        //----------------------------------------------------
        // Paste Position
        //----------------------------------------------------
        GVL_1.DATA_RB_B.X_POS[GVL.HMI_B_PointNoSelected] := GVL.B_PointClipboardX;

        GVL_1.DATA_RB_B.Y_POS[GVL.HMI_B_PointNoSelected] := GVL.B_PointClipboardY;

        GVL_1.DATA_RB_B.Z_POS[GVL.HMI_B_PointNoSelected] := GVL.B_PointClipboardZ;

        GVL_1.DATA_RB_B.R_POS[GVL.HMI_B_PointNoSelected] := GVL.B_PointClipboardR;


//         //----------------------------------------------------
//         // Đồng thời cập nhật vùng Edit để HMI hiển thị
//         // ngay dữ liệu vừa Paste
//         //----------------------------------------------------
//         GVL.HMI_B_Edit_PointNo := GVL.HMI_B_PointNoSelected;
// 
//         GVL.HMI_B_Edit_Pos_Name := GVL.B_PointClipboardName;
// 
//         GVL.HMI_B_Edit_Pos_X := GVL.B_PointClipboardX;
// 
//         GVL.HMI_B_Edit_Pos_Y := GVL.B_PointClipboardY;
// 
//         GVL.HMI_B_Edit_Pos_Z := GVL.B_PointClipboardZ;
// 
//         GVL.HMI_B_Edit_Pos_R := GVL.B_PointClipboardR;

    END_IF;

    //--------------------------------------------------------
    // Không xóa Clipboard.
    //
    // Nhờ vậy có thể:
    // Copy P10 → Paste P20 → Paste P21 → Paste P22...
    //--------------------------------------------------------

    GVL.HMI_B_EditPointReq := 0;

END_IF;

//============================================================
// DELETE ALL POINTS
//
// HMI_A_EditPointReq = 27
//
// Xóa toàn bộ Point Database.
//============================================================

Delete_all_point_B(IN := GVL.HMI_B_EditPointReq_Arr[7], PT := T#2S);
IF Delete_all_point_B.Q THEN

    FOR iPoint := 1 TO 500 DO

        //----------------------------------------------------
        // Clear Name
        //----------------------------------------------------
        GVL_1.Point_Name_B[iPoint] := '';

        //----------------------------------------------------
        // Clear Position
        //----------------------------------------------------
        GVL_1.DATA_RB_B.X_POS[iPoint] := 0.0;
        GVL_1.DATA_RB_B.Y_POS[iPoint] := 0.0;
        GVL_1.DATA_RB_B.Z_POS[iPoint] := 0.0;
        GVL_1.DATA_RB_B.R_POS[iPoint] := 0.0;

    END_FOR;


    //--------------------------------------------------------
    // Clear vùng Edit trên HMI
    //--------------------------------------------------------
    GVL.HMI_B_Edit_PointNo  := 0;
    GVL.HMI_B_Edit_Pos_Name := '';

    GVL.HMI_B_Edit_Pos_X := 0.0;
    GVL.HMI_B_Edit_Pos_Y := 0.0;
    GVL.HMI_B_Edit_Pos_Z := 0.0;
    GVL.HMI_B_Edit_Pos_R := 0.0;


    //--------------------------------------------------------
    // Reset Point đang chọn
    //--------------------------------------------------------
    GVL.HMI_B_PointNoSelected := 0;


    //--------------------------------------------------------
    // Em khuyên KHÔNG xóa Clipboard.
    //
    // Nếu Delete All nhầm, dữ liệu Point vừa Copy vẫn còn
    // và có thể Paste lại.
    //--------------------------------------------------------

    GVL.HMI_B_EditPointReq := 0;
	GVL.HMI_B_EditPointReq_Arr[7] := FALSE;

END_IF;
END_ACTION

END_PROGRAM

// Just_Motion_Control_x86_64_Linux_SM_WV/Application/FC_/RBA/F_EvalCondRowFromEdit_A
FUNCTION F_EvalCondRowFromEdit_A : BOOL
VAR_INPUT
	RowNo : INT;
END_VAR
VAR
	actualValue : DINT;
END_VAR

IF (RowNo < 1) OR (RowNo > 10) THEN
    F_EvalCondRowFromEdit_A := FALSE;
    RETURN;
END_IF;

IF NOT GVL.HMI_A_CondEditRowEnable[RowNo] THEN
    F_EvalCondRowFromEdit_A := TRUE;
    RETURN;
END_IF;

// Đọc giá trị thực tế hiện tại
actualValue := F_GetCondValue_A(
    Source := GVL.HMI_A_CondEditSource[RowNo],
    Index  := GVL.HMI_A_CondEditIndex[RowNo]
);

// Lưu actual value để HMI hiển thị
GVL.HMI_A_CondMonActualValue[RowNo] := actualValue;

// So sánh theo operator
CASE GVL.HMI_A_CondEditOperator[RowNo] OF
    1: F_EvalCondRowFromEdit_A := actualValue = GVL.HMI_A_CondEditSetValue[RowNo];
    2: F_EvalCondRowFromEdit_A := actualValue <> GVL.HMI_A_CondEditSetValue[RowNo];
    3: F_EvalCondRowFromEdit_A := actualValue >  GVL.HMI_A_CondEditSetValue[RowNo];
    4: F_EvalCondRowFromEdit_A := actualValue >= GVL.HMI_A_CondEditSetValue[RowNo];
    5: F_EvalCondRowFromEdit_A := actualValue <  GVL.HMI_A_CondEditSetValue[RowNo];
    6: F_EvalCondRowFromEdit_A := actualValue <= GVL.HMI_A_CondEditSetValue[RowNo];
ELSE
    F_EvalCondRowFromEdit_A := FALSE;
END_CASE;

END_FUNCTION

// Just_Motion_Control_x86_64_Linux_SM_WV/Application/FC_/RBB/F_EvalCondRowFromEdit_B
FUNCTION F_EvalCondRowFromEdit_B : BOOL
VAR_INPUT
	RowNo : INT;
END_VAR
VAR
	actualValue : DINT;
END_VAR

IF (RowNo < 1) OR (RowNo > 10) THEN
    F_EvalCondRowFromEdit_B := FALSE;
    RETURN;
END_IF;

IF NOT GVL.HMI_B_CondEditRowEnable[RowNo] THEN
    F_EvalCondRowFromEdit_B := TRUE;
    RETURN;
END_IF;

// Đọc giá trị thực tế hiện tại
actualValue := F_GetCondValue_B(
    Source := GVL.HMI_B_CondEditSource[RowNo],
    Index  := GVL.HMI_B_CondEditIndex[RowNo]
);

// Lưu actual value để HMI hiển thị
GVL.HMI_B_CondMonActualValue[RowNo] := actualValue;

// So sánh theo operator
CASE GVL.HMI_B_CondEditOperator[RowNo] OF
    1: F_EvalCondRowFromEdit_B := actualValue = GVL.HMI_B_CondEditSetValue[RowNo];
    2: F_EvalCondRowFromEdit_B := actualValue <> GVL.HMI_B_CondEditSetValue[RowNo];
    3: F_EvalCondRowFromEdit_B := actualValue >  GVL.HMI_B_CondEditSetValue[RowNo];
    4: F_EvalCondRowFromEdit_B := actualValue >= GVL.HMI_B_CondEditSetValue[RowNo];
    5: F_EvalCondRowFromEdit_B := actualValue <  GVL.HMI_B_CondEditSetValue[RowNo];
    6: F_EvalCondRowFromEdit_B := actualValue <= GVL.HMI_B_CondEditSetValue[RowNo];
ELSE
    F_EvalCondRowFromEdit_B := FALSE;
END_CASE;

END_FUNCTION

// Just_Motion_Control_x86_64_Linux_SM_WV/Application/PRG_ROBOT/POU_HOMING
PROGRAM POU_HOMING
VAR
	MC_GroupStop_RBA, MC_GroupStop_RBB : MC_GroupStop;
	MC_Stop_A0: MC_Stop;
	MC_Stop_A1: MC_Stop;
	MC_Stop_A2: MC_Stop;
	MC_Stop_A3: MC_Stop;
	MC_GroupSetPosition_RB1: MC_GroupSetPosition;
	Origin_Pos_A: SM3_Robotics.SMC_POS_REF;
	MC_GroupSetPosition_RB2: MC_GroupSetPosition;
	Origin_Pos_B: SM3_Robotics.SMC_POS_REF;
	MC_Stop_B0: MC_Stop;
	MC_Stop_B2: MC_Stop;
	MC_Stop_B1: MC_Stop;
	MC_Stop_B3: MC_Stop;
	MC_Home_A0: MC_Home;
	MC_Home_A1: MC_Home;
	MC_Home_A2: MC_Home;
	MC_Home_A3: MC_Home;
	MC_Home_B0: MC_Home;
	MC_Home_B1: MC_Home;
	MC_Home_B2: MC_Home;
	MC_Home_B3: MC_Home;
	MC_Power_za: MC_Power;
	MC_Jog_za: MC_Jog;
	MC_Power_ZB: MC_Power;
	MC_Jog_ZB: MC_Jog;
	SMC_SetSoftwareLimits_A0: SMC_SetSoftwareLimits;
	SMC_SetSoftwareLimits_A1: SMC_SetSoftwareLimits;
	SMC_SetSoftwareLimits_A2: SMC_SetSoftwareLimits;
	SMC_SetSoftwareLimits_A3: SMC_SetSoftwareLimits;
	SMC_SetSoftwareLimits_B0: SMC_SetSoftwareLimits;
	SMC_SetSoftwareLimits_B1: SMC_SetSoftwareLimits;
	SMC_SetSoftwareLimits_B2: SMC_SetSoftwareLimits;
	SMC_SetSoftwareLimits_B3: SMC_SetSoftwareLimits;
	
	MC_ReadError_A0: MC_ReadAxisError;
	MC_ReadError_A1: MC_ReadAxisError;
	MC_ReadError_A2: MC_ReadAxisError;
	MC_ReadError_A3: MC_ReadAxisError;
	MC_ReadError_B0: MC_ReadAxisError;
	MC_ReadError_B1: MC_ReadAxisError;
	MC_ReadError_B2: MC_ReadAxisError;
	MC_ReadError_B3: MC_ReadAxisError;
	
END_VAR
VAR
	Bit_Stop, BitStop_Tor_A, BitStop_Tor_B, BitStop_TorDiff_A, BitStop_TorDiff_B, BitStop_Error_Axis_RB_A, BitStop_Error_Axis_RB_B : BOOL;	
	//EMG AT %IX1.1 : BOOL;
	
	// Home Z 
	D_HomeZ_RB1, D_HomeZ_RB2 : INT;
	//SS_DOG_Z1 AT %IX1.3 : BOOL;
	//SS_DOG_Z2 AT %IX1.2 : BOOL;
	R_TRIG_Z1, R_TRIG_Z2 : R_TRIG;
	Homing_Z1, Homing_Z2, Home_Done_Z1, Home_Done_Z2 : BOOL;
END_VAR

VAR // SETLMIT
	ENABLE_POWER_A,DISABLE_POWER_A, ENABLE_POWER_B, DISABLE_POWER_B : BYTE;
	
END_VAR
VAR
	TORQUE_ACT_A0 AT %IW40 : INT;
	TORQUE_ACT_A1 AT %IW48 : INT;
	TORQUE_ACT_A2 AT %IW56 : INT;
	TORQUE_ACT_A3 AT %IW64 : INT;
	TORQUE_ACT_B0 AT %IW72 : INT;
	TORQUE_ACT_B1 AT %IW80 : INT;
	TORQUE_ACT_B2 AT %IW88 : INT;
	TORQUE_ACT_B3 AT %IW96 : INT;
	TORQUE_LIMIT_A0, TORQUE_LIMIT_A1, TORQUE_LIMIT_A2, TORQUE_LIMIT_A3 : INT;
	TORQUE_LIMIT_B0, TORQUE_LIMIT_B1, TORQUE_LIMIT_B2, TORQUE_LIMIT_B3 : INT;
	
END_VAR

//namnv0804
VAR
	VEL_ACT_A0 AT %ID19 : DINT;
	VEL_ACT_A1 AT %ID23 : DINT;
	VEL_ACT_A2 AT %ID27 : DINT;
	VEL_ACT_A3 AT %ID31 : DINT;
	VEL_ACT_B0 AT %ID35 : DINT;
	VEL_ACT_B1 AT %ID39 : DINT;
	VEL_ACT_B2 AT %ID43 : DINT;
	VEL_ACT_B3 AT %ID47 : DINT;
	
	VEL_SET_A0 AT %QD118 : DINT;
	VEL_SET_A1 AT %QD122 : DINT;
	VEL_SET_A2 AT %QD126 : DINT;
	VEL_SET_A3 AT %QD130 : DINT;
	VEL_SET_B0 AT %QD134 : DINT;
	VEL_SET_B1 AT %QD138 : DINT;
	VEL_SET_B2 AT %QD142 : DINT;
	VEL_SET_B3 AT %QD146 : DINT;
	
	TorqueDiff_RB_A0, TorqueDiff_RB_A1, TorqueDiff_RB_A2, TorqueDiff_RB_A3 : FB_TorqueDiff;
	TorqueDiff_RB_B0, TorqueDiff_RB_B1, TorqueDiff_RB_B2, TorqueDiff_RB_B3 : FB_TorqueDiff;
	TORQUE_DIFF_LIMIT_B0, TORQUE_DIFF_LIMIT_B1, TORQUE_DIFF_LIMIT_B2, TORQUE_DIFF_LIMIT_B3 : INT;
	TORQUE_DIFF_MAX_A0, TORQUE_DIFF_MAX_A1, TORQUE_DIFF_MAX_A2, TORQUE_DIFF_MAX_A3 : INT;
	TORQUE_DIFF_MAX_B0, TORQUE_DIFF_MAX_B1, TORQUE_DIFF_MAX_B2, TORQUE_DIFF_MAX_B3 : INT;
	TORQUE_DIFF_MIN_A0, TORQUE_DIFF_MIN_A1, TORQUE_DIFF_MIN_A2, TORQUE_DIFF_MIN_A3 : INT;
	TORQUE_DIFF_MIN_B0, TORQUE_DIFF_MIN_B1, TORQUE_DIFF_MIN_B2, TORQUE_DIFF_MIN_B3 : INT;
	
	VEL_MAX_A0, VEL_MAX_A1, VEL_MAX_A2, VEL_MAX_A3 : DINT;
	VEL_MAX_B0, VEL_MAX_B1, VEL_MAX_B2, VEL_MAX_B3 : DINT;
	
	VEL_SET_MAX_A0, VEL_SET_MAX_A1, VEL_SET_MAX_A2, VEL_SET_MAX_A3 : DINT;
	VEL_SET_MAX_B0, VEL_SET_MAX_B1, VEL_SET_MAX_B2, VEL_SET_MAX_B3 : DINT;
	Vel_Act_Per_Vel_Set_A0, Vel_Act_Per_Vel_Set_A1, Vel_Act_Per_Vel_Set_A2, Vel_Act_Per_Vel_Set_A3: INT;
	Vel_Act_Per_Vel_Set_B0, Vel_Act_Per_Vel_Set_B1, Vel_Act_Per_Vel_Set_B2, Vel_Act_Per_Vel_Set_B3: INT;
	Torque_arr_A0 : ARRAY[0..20000] OF INT;
	i_A0 : INT := 0;
END_VAR
VAR // added by the converter: edge detectors and wires of the graphical bodies
    _w1, _w2, _w3, _w4, _w5, _w6, _w7, _w8 : LREAL;
END_VAR

// namnv3103
// TORQUE_LIMIT_A0:= 3600;
// TORQUE_LIMIT_A1:= 2500;
// TORQUE_LIMIT_A2:= 2000;
// TORQUE_LIMIT_A3:= 2000;
// 
// TORQUE_LIMIT_B0:= 3600;
// TORQUE_LIMIT_B1:= 2500;
// TORQUE_LIMIT_B2:= 2000;
// TORQUE_LIMIT_B3:= 2000;

TORQUE_LIMIT_A0:= GVL.Pro4_.Auto.TORQUE_LIMIT_SET_A0;
TORQUE_LIMIT_A1:= GVL.Pro4_.Auto.TORQUE_LIMIT_SET_A1;
TORQUE_LIMIT_A2:= GVL.Pro4_.Auto.TORQUE_LIMIT_SET_A2;
TORQUE_LIMIT_A3:= GVL.Pro4_.Auto.TORQUE_LIMIT_SET_A3;

TORQUE_LIMIT_B0:= GVL.Pro4_.Auto.TORQUE_LIMIT_SET_B0;
TORQUE_LIMIT_B1:= GVL.Pro4_.Auto.TORQUE_LIMIT_SET_B1;
TORQUE_LIMIT_B2:= GVL.Pro4_.Auto.TORQUE_LIMIT_SET_B2;
TORQUE_LIMIT_B3:= GVL.Pro4_.Auto.TORQUE_LIMIT_SET_B3;

IF GVL.Reset_Torque_Max THEN
	GVL.Torque_Max.A0 := 0;
	GVL.Torque_Max.A1 := 0;
	GVL.Torque_Max.A2 := 0;
	GVL.Torque_Max.A3 := 0;
	GVL.Torque_Max.B0 := 0;
	GVL.Torque_Max.B1 := 0;
	GVL.Torque_Max.B2 := 0;
	GVL.Torque_Max.B3 := 0;
	TORQUE_DIFF_MAX_A0 := 0;
	TORQUE_DIFF_MAX_A1 := 0;
	TORQUE_DIFF_MAX_A2 := 0;
	TORQUE_DIFF_MAX_A3 := 0;
	TORQUE_DIFF_MAX_B0 := 0;
	TORQUE_DIFF_MAX_B1 := 0;
	TORQUE_DIFF_MAX_B2 := 0;
	TORQUE_DIFF_MAX_B3 := 0;
	VEL_MAX_A0 := 0;
	VEL_MAX_A1 := 0;
	VEL_MAX_A2 := 0;
	VEL_MAX_A3 := 0;
	VEL_MAX_B0 := 0;
	VEL_MAX_B1 := 0;
	VEL_MAX_B2 := 0;
	VEL_MAX_B3 := 0;
	VEL_SET_MAX_A0 := 0;
END_IF
GVL.Torque_Max.A0 := MAX(ABS(TORQUE_ACT_A0), GVL.Torque_Max.A0);
GVL.Torque_Max.A1 := MAX(ABS(TORQUE_ACT_A1), GVL.Torque_Max.A1);
GVL.Torque_Max.A2 := MAX(ABS(TORQUE_ACT_A2), GVL.Torque_Max.A2);
GVL.Torque_Max.A3 := MAX(ABS(TORQUE_ACT_A3), GVL.Torque_Max.A3);

GVL.Torque_Max.B0 := MAX(ABS(TORQUE_ACT_B0), GVL.Torque_Max.B0);
GVL.Torque_Max.B1 := MAX(ABS(TORQUE_ACT_B1), GVL.Torque_Max.B1);
GVL.Torque_Max.B2 := MAX(ABS(TORQUE_ACT_B2), GVL.Torque_Max.B2);
GVL.Torque_Max.B3 := MAX(ABS(TORQUE_ACT_B3), GVL.Torque_Max.B3);

// IF (ABS(TORQUE_ACT_A0) > TORQUE_LIMIT_A0) OR (ABS(TORQUE_ACT_A1) > TORQUE_LIMIT_A1) OR (ABS(TORQUE_ACT_A2) > TORQUE_LIMIT_A2) OR (ABS(TORQUE_ACT_A3) > TORQUE_LIMIT_A3) THEN
// 	BitStop_Tor_A := TRUE;
// ELSE
// 	BitStop_Tor_A := FALSE;
// END_IF
// 
// IF (ABS(TORQUE_ACT_B0) > TORQUE_LIMIT_B0) OR (ABS(TORQUE_ACT_B1) > TORQUE_LIMIT_B1) OR (ABS(TORQUE_ACT_B2) > TORQUE_LIMIT_B2) OR (ABS(TORQUE_ACT_B3) > TORQUE_LIMIT_B3) THEN
// 	BitStop_Tor_B := TRUE;
// ELSE
// 	BitStop_Tor_B := FALSE;
// END_IF

//namnv0804

VEL_MAX_A0 := MAX(VEL_MAX_A0, ABS(VEL_ACT_A0));
VEL_MAX_A1 := MAX(VEL_MAX_A1, ABS(VEL_ACT_A1));
VEL_MAX_A2 := MAX(VEL_MAX_A2, ABS(VEL_ACT_A2));
VEL_MAX_A3 := MAX(VEL_MAX_A3, ABS(VEL_ACT_A3));
VEL_MAX_B0 := MAX(VEL_MAX_B0, ABS(VEL_ACT_B0));
VEL_MAX_B1 := MAX(VEL_MAX_B1, ABS(VEL_ACT_B1));
VEL_MAX_B2 := MAX(VEL_MAX_B2, ABS(VEL_ACT_B2));
VEL_MAX_B3 := MAX(VEL_MAX_B3, ABS(VEL_ACT_B3));
VEL_SET_MAX_A0 := MAX(VEL_SET_MAX_A0, ABS(VEL_SET_A0));
Vel_Act_Per_Vel_Set_A0 := LREAL_TO_INT(
    (DINT_TO_LREAL(VEL_ACT_A0) * 100.0) / DINT_TO_LREAL(VEL_SET_A0)
);
Vel_Act_Per_Vel_Set_A1 := LREAL_TO_INT(
    (DINT_TO_LREAL(VEL_ACT_A1) * 100.0) / DINT_TO_LREAL(VEL_SET_A1)
);
Vel_Act_Per_Vel_Set_A2 := LREAL_TO_INT(
    (DINT_TO_LREAL(VEL_ACT_A2) * 100.0) / DINT_TO_LREAL(VEL_SET_A2)
);
Vel_Act_Per_Vel_Set_A3 := LREAL_TO_INT(
    (DINT_TO_LREAL(VEL_ACT_A3) * 100.0) / DINT_TO_LREAL(VEL_SET_A3)
);
Vel_Act_Per_Vel_Set_B0 := LREAL_TO_INT(
    (DINT_TO_LREAL(VEL_ACT_B0) * 100.0) / DINT_TO_LREAL(VEL_SET_B0)
);
Vel_Act_Per_Vel_Set_B1 := LREAL_TO_INT(
    (DINT_TO_LREAL(VEL_ACT_B1) * 100.0) / DINT_TO_LREAL(VEL_SET_B1)
);
Vel_Act_Per_Vel_Set_B2 := LREAL_TO_INT(
    (DINT_TO_LREAL(VEL_ACT_B2) * 100.0) / DINT_TO_LREAL(VEL_SET_B2)
);
Vel_Act_Per_Vel_Set_B3 := LREAL_TO_INT(
    (DINT_TO_LREAL(VEL_ACT_B3) * 100.0) / DINT_TO_LREAL(VEL_SET_B3)
);

TorqueDiff_RB_A0(
	Enable := TRUE,
	TorqueNow := TORQUE_ACT_A0,
	PercentVel := Vel_Act_Per_Vel_Set_A0,
	Threshold := 400,
	CycleTime_s := 0.01
);
TorqueDiff_RB_A1(
	Enable := TRUE,
	TorqueNow := TORQUE_ACT_A1,
	PercentVel := Vel_Act_Per_Vel_Set_A1,
	Threshold := 500,
	CycleTime_s := 0.01
);
TorqueDiff_RB_A2(
	Enable := TRUE,
	TorqueNow := TORQUE_ACT_A2,
	PercentVel := Vel_Act_Per_Vel_Set_A2,
	Threshold := 500,
	CycleTime_s := 0.01
);
TorqueDiff_RB_A3(
	Enable := TRUE,
	TorqueNow := TORQUE_ACT_A3,
	PercentVel := Vel_Act_Per_Vel_Set_A3,
	Threshold := 100,
	CycleTime_s := 0.01
);

TorqueDiff_RB_B0(
	Enable := TRUE,
	TorqueNow := TORQUE_ACT_B0,
	PercentVel := Vel_Act_Per_Vel_Set_B0,
	Threshold := 500,
	CycleTime_s := 0.01
);
TorqueDiff_RB_B1(
	Enable := TRUE,
	TorqueNow := TORQUE_ACT_B1,
	PercentVel := Vel_Act_Per_Vel_Set_B1,
	Threshold := 500,
	CycleTime_s := 0.01
);
TorqueDiff_RB_B2(
	Enable := TRUE,
	TorqueNow := TORQUE_ACT_B2,
	PercentVel := Vel_Act_Per_Vel_Set_B2,
	Threshold := 500,
	CycleTime_s := 0.01
);
TorqueDiff_RB_B3(
	Enable := TRUE,
	TorqueNow := TORQUE_ACT_B3,
	PercentVel := Vel_Act_Per_Vel_Set_B3,
	Threshold := 100,
	CycleTime_s := 0.01
);

TORQUE_DIFF_MAX_A0 := MAX(TORQUE_DIFF_MAX_A0, TorqueDiff_RB_A0.AbsDeltaTorque);
TORQUE_DIFF_MAX_A1 := MAX(TORQUE_DIFF_MAX_A1, TorqueDiff_RB_A1.AbsDeltaTorque);
TORQUE_DIFF_MAX_A2 := MAX(TORQUE_DIFF_MAX_A2, TorqueDiff_RB_A2.AbsDeltaTorque);
TORQUE_DIFF_MAX_A3 := MAX(TORQUE_DIFF_MAX_A3, TorqueDiff_RB_A3.AbsDeltaTorque);
TORQUE_DIFF_MAX_B0 := MAX(TORQUE_DIFF_MAX_B0, TorqueDiff_RB_B0.AbsDeltaTorque);
TORQUE_DIFF_MAX_B1 := MAX(TORQUE_DIFF_MAX_B1, TorqueDiff_RB_B1.AbsDeltaTorque);
TORQUE_DIFF_MAX_B2 := MAX(TORQUE_DIFF_MAX_B2, TorqueDiff_RB_B2.AbsDeltaTorque);
TORQUE_DIFF_MAX_B3 := MAX(TORQUE_DIFF_MAX_B3, TorqueDiff_RB_B3.AbsDeltaTorque);

IF (TorqueDiff_RB_A0.Alarm) OR (TorqueDiff_RB_A1.Alarm) OR (TorqueDiff_RB_A2.Alarm) OR (TorqueDiff_RB_A3.Alarm) THEN
	BitStop_TorDiff_A := TRUE;
ELSE
	BitStop_TorDiff_A := FALSE;
END_IF

IF (TorqueDiff_RB_B0.Alarm) OR (TorqueDiff_RB_B1.Alarm) OR (TorqueDiff_RB_B2.Alarm) OR (TorqueDiff_RB_B3.Alarm) THEN
	BitStop_TorDiff_B := TRUE;
ELSE
	BitStop_TorDiff_B := FALSE;
END_IF


ACT_HOMING();
ACT_STOP();
ACT_Home_Z();
ACT_SETLIMIT();
ACT_ERROR(); //namnv0304

//Origin_Pos_A.c.X := 550;
//Origin_Pos_B.c.X := 0;
//Origin_Pos_B.a.a0 := 0;

ACTION ACT_ERROR:
MC_ReadError_A0(Axis := A0, Enable := A0.bError); // MC_ReadAxisError
MC_ReadError_B0(Axis := B0, Enable := B0.bError); // MC_ReadAxisError
MC_ReadError_A2(Axis := A2, Enable := A2.bError); // MC_ReadAxisError
MC_ReadError_B1(Axis := B1, Enable := B1.bError); // MC_ReadAxisError
MC_ReadError_A3(Axis := A3, Enable := A3.bError); // MC_ReadAxisError
MC_ReadError_A1(Axis := A1, Enable := A1.bError); // MC_ReadAxisError
MC_ReadError_B2(Axis := B2, Enable := B2.bError); // MC_ReadAxisError
MC_ReadError_B3(Axis := B3, Enable := B3.bError); // MC_ReadAxisError
END_ACTION

ACTION ACT_Home_Z:
IF GVL.RB_A.M3 AND GVL.RB_A.Manual AND MC_Power_za.Status THEN
	Homing_Z1 := TRUE;
ELSIF NOT GVL.X[9] OR NOT MC_Power_za.Status THEN
	Homing_Z1 := FALSE;
END_IF
MC_Home_A2.Execute := GVL.RB_A.ORG_M3;
/// PRocess
IF Homing_Z1 THEN
CASE D_HomeZ_RB1 OF
	0:
		IF  GVL.X[3] THEN
			MC_Jog_za.Velocity := 10;
			MC_Jog_za.JogBackward := TRUE;
		ELSE
			MC_Jog_za.JogBackward := FALSE;
			D_HomeZ_RB1 := D_HomeZ_RB1 + 10;
		END_IF
	10:
		IF NOT GVL.X[3] THEN
			MC_Jog_za.Velocity := 5;
			MC_Jog_za.JogForward := TRUE;
		ELSE
			D_HomeZ_RB1 := D_HomeZ_RB1 + 5;
		END_IF
	15:
		IF GVL.X[3] THEN
			MC_Jog_za.JogForward := FALSE;
			D_HomeZ_RB1 := D_HomeZ_RB1 + 5;
		END_IF
	20:
		MC_Jog_za.JogForward := FALSE;
		MC_Jog_za.JogBackward := FALSE;
		MC_Home_A2.Execute := TRUE;
		D_HomeZ_RB1 := D_HomeZ_RB1 + 10;
	30:
		IF MC_Home_A2.Done OR MC_Home_A2.Busy THEN
			MC_Home_A2.Execute := FALSE;
			D_HomeZ_RB1 := D_HomeZ_RB1 + 10;
		ELSIF MC_Home_A2.Error THEN
			D_HomeZ_RB1 := 900;
		END_IF					
	40:	
		D_HomeZ_RB1 := D_HomeZ_RB1 + 10;	
	50:
		D_HomeZ_RB1 := 900;
///////////////////////////////////////// Process Done ////////////////////////////////////
	900:
		Homing_Z1 := FALSE;
END_CASE
ELSE
	MC_Jog_za.JogForward := FALSE;
	MC_Jog_za.JogBackward := FALSE;
	D_HomeZ_RB1 := 0;
END_IF



///// Home Z2 robot B

IF GVL.RB_B.M3 AND GVL.RB_B.Manual AND MC_Power_zB.Status THEN
	Homing_Z2 := TRUE;
ELSIF NOT GVL.X[9] OR NOT MC_Power_ZB.Status THEN
	Homing_Z2 := FALSE;
END_IF
MC_Home_B2.Execute := GVL.RB_B.ORG_M3;
/// PRocess
IF Homing_Z2 THEN
CASE D_HomeZ_RB2 OF
	0:
		IF  GVL.X[2] THEN
			MC_Jog_ZB.Velocity := 10;
			MC_Jog_ZB.JogBackward := TRUE;
		ELSE
			MC_Jog_ZB.JogBackward := FALSE;
			D_HomeZ_RB2 := D_HomeZ_RB2 + 10;
		END_IF
	10:
		IF NOT GVL.X[2] THEN
			MC_Jog_ZB.Velocity := 5;
			MC_Jog_ZB.JogForward := TRUE;
		ELSE
			D_HomeZ_RB2 := D_HomeZ_RB2 + 5;
		END_IF
	15:
		IF GVL.X[2] THEN
			MC_Jog_ZB.JogForward := FALSE;
			D_HomeZ_RB2 := D_HomeZ_RB2 + 5;
		END_IF
	20:
		MC_Jog_ZB.JogForward := FALSE;
		MC_Jog_ZB.JogBackward := FALSE;
		MC_Home_b2.Execute := TRUE;
		D_HomeZ_RB2 := D_HomeZ_RB2 + 10;
	30:
		IF MC_Home_b2.Done OR MC_Home_b2.Busy THEN
			MC_Home_b2.Execute := FALSE;
			D_HomeZ_RB2 := D_HomeZ_RB2 + 10;
		ELSIF MC_Home_b2.Error THEN
			D_HomeZ_RB2 := 900;
		END_IF					
	40:	
		D_HomeZ_RB2 := D_HomeZ_RB2 + 10;	
	50:
		D_HomeZ_RB2 := 900;
///////////////////////////////////////// Process Done ////////////////////////////////////
	900:
		Homing_Z2 := FALSE;
END_CASE
ELSE
	MC_Jog_ZB.JogForward := FALSE;
	MC_Jog_ZB.JogBackward := FALSE;
	D_HomeZ_RB2 := 0;
END_IF
END_ACTION

ACTION ACT_HOMING:
MC_GroupSetPosition_RB1(AxisGroup := SCARA_A, Position := Origin_Pos_A, CoordSystem := GVL.RB_A.COORD); // MC_GroupSetPosition
MC_GroupSetPosition_RB2(AxisGroup := SCARA_B, Position := Origin_Pos_B, CoordSystem := GVL.RB_B.COORD); // MC_GroupSetPosition
MC_Power_ZB(Axis := B2); // MC_Power
MC_Jog_za(Axis := A2, Acceleration := 500, Deceleration := 500, Jerk := 1000); // MC_Jog
MC_Jog_ZB(Axis := B2, Acceleration := 500, Deceleration := 500, Jerk := 1000); // MC_Jog
MC_Home_B2(Axis := B2, Position := 0); // MC_Home
MC_Home_A2(Axis := A2, Position := 0); // MC_Home
MC_Home_B1(Axis := B1, Execute := GVL.RB_B.ORG_M2, Position := 0); // MC_Home
MC_Power_za(Axis := A2); // MC_Power
MC_Home_A1(Axis := A1, Execute := GVL.RB_A.ORG_M2, Position := 0); // MC_Home
MC_Home_B3(Axis := B3, Execute := GVL.RB_B.ORG_M4, Position := 0); // MC_Home
MC_Home_A3(Axis := A3, Execute := GVL.RB_A.ORG_M4, Position := 0); // MC_Home
MC_Home_B0(Axis := B0, Execute := GVL.RB_B.ORG_M1, Position := 0); // MC_Home
MC_Home_A0(Axis := A0, Execute := GVL.RB_A.ORG_M1, Position := 0); // MC_Home
MC_Stop_B0(Axis := B0, Deceleration := 100, Jerk := 0); // MC_Stop
MC_Stop_B1(Axis := B1, Deceleration := 100, Jerk := 0); // MC_Stop
MC_Stop_B2(Axis := B2, Deceleration := 100, Jerk := 0); // MC_Stop
MC_Stop_B3(Axis := B3, Deceleration := 100, Jerk := 0); // MC_Stop
MC_Stop_A0(Axis := A0, Deceleration := 100, Jerk := 0); // MC_Stop
MC_Stop_A3(Axis := A3, Deceleration := 100, Jerk := 0); // MC_Stop
MC_Stop_A2(Axis := A2, Deceleration := 100, Jerk := 0); // MC_Stop
MC_Stop_A1(Axis := A1, Deceleration := 100, Jerk := 0); // MC_Stop
END_ACTION

ACTION ACT_SETLIMIT:
_w1 := TO_LREAL(GVL_1.DATA_RB_A.LIMIT_M1_BW);
_w2 := TO_LREAL(GVL_1.DATA_RB_B.LIMIT_M2_FW);
_w3 := TO_LREAL(GVL_1.DATA_RB_B.LIMIT_M2_BW);
SMC_SetSoftwareLimits_A1(
    Axis := A1,
    SWL_Positive := TO_LREAL(GVL_1.DATA_RB_A.LIMIT_M2_FW),
    SWL_Negative := TO_LREAL(GVL_1.DATA_RB_A.LIMIT_M2_BW),
    SWL_Error_Deceleration := 1000,
    SWL_Error_MaxDistance := 10); // SMC_SetSoftwareLimits
_w4 := TO_LREAL(GVL_1.DATA_RB_B.LIMIT_M3_FW);
_w5 := TO_LREAL(GVL_1.DATA_RB_B.LIMIT_M3_BW);
SMC_SetSoftwareLimits_A2(
    Axis := A2,
    SWL_Positive := TO_LREAL(GVL_1.DATA_RB_A.LIMIT_M3_FW),
    SWL_Negative := TO_LREAL(GVL_1.DATA_RB_A.LIMIT_M3_BW),
    SWL_Error_Deceleration := 1000,
    SWL_Error_MaxDistance := 10); // SMC_SetSoftwareLimits
_w6 := TO_LREAL(GVL_1.DATA_RB_B.LIMIT_M4_FW);
_w7 := TO_LREAL(GVL_1.DATA_RB_B.LIMIT_M4_BW);
_w8 := TO_LREAL(GVL_1.DATA_RB_B.LIMIT_M1_FW);
SMC_SetSoftwareLimits_A3(
    Axis := A3,
    SWL_Positive := TO_LREAL(GVL_1.DATA_RB_A.LIMIT_M4_FW),
    SWL_Negative := TO_LREAL(GVL_1.DATA_RB_A.LIMIT_M4_BW),
    SWL_Error_Deceleration := 1000,
    SWL_Error_MaxDistance := 10); // SMC_SetSoftwareLimits
SMC_SetSoftwareLimits_B0(
    Axis := B0,
    SWL_Positive := _w8,
    SWL_Negative := TO_LREAL(GVL_1.DATA_RB_B.LIMIT_M1_BW),
    SWL_Error_Deceleration := 1000,
    SWL_Error_MaxDistance := 10); // SMC_SetSoftwareLimits
SMC_SetSoftwareLimits_B2(
    Axis := B2,
    SWL_Positive := _w4,
    SWL_Negative := _w5,
    SWL_Error_Deceleration := 1000,
    SWL_Error_MaxDistance := 10); // SMC_SetSoftwareLimits
SMC_SetSoftwareLimits_B3(
    Axis := B3,
    SWL_Positive := _w6,
    SWL_Negative := _w7,
    SWL_Error_Deceleration := 1000,
    SWL_Error_MaxDistance := 10); // SMC_SetSoftwareLimits
SMC_SetSoftwareLimits_A0(
    Axis := A0,
    SWL_Positive := TO_LREAL(GVL_1.DATA_RB_A.LIMIT_M1_FW),
    SWL_Negative := _w1,
    SWL_Error_Deceleration := 1000,
    SWL_Error_MaxDistance := 10); // SMC_SetSoftwareLimits
SMC_SetSoftwareLimits_B1(
    Axis := B1,
    SWL_Positive := _w2,
    SWL_Negative := _w3,
    SWL_Error_Deceleration := 1000,
    SWL_Error_MaxDistance := 10); // SMC_SetSoftwareLimits
END_ACTION

ACTION ACT_STOP:
IF (MC_ReadError_A0.AxisError OR MC_ReadError_A1.AxisError OR MC_ReadError_A2.AxisError OR MC_ReadError_A3.AxisError) 
OR (MC_ReadError_A0.Error OR MC_ReadError_A1.Error OR MC_ReadError_A2.Error OR MC_ReadError_A3.Error)
OR A0.bError OR A1.bError OR A2.bError OR A3.bError THEN
	BitStop_Error_Axis_RB_A := TRUE;
ELSE
	BitStop_Error_Axis_RB_A := FALSE;
END_IF

IF (MC_ReadError_B0.AxisError OR MC_ReadError_B1.AxisError OR MC_ReadError_B2.AxisError OR MC_ReadError_B3.AxisError) 
OR (MC_ReadError_B0.Error OR MC_ReadError_B1.Error OR MC_ReadError_B2.Error OR MC_ReadError_B3.Error) 
OR B0.bError OR B1.bError OR B2.bError OR B3.bError THEN
	BitStop_Error_Axis_RB_B := TRUE;
ELSE
	BitStop_Error_Axis_RB_B := FALSE;
END_IF

IF Bit_Stop = TRUE OR NOT GVL.X[9] OR BitStop_Tor_A OR BitStop_Error_Axis_RB_A 
OR GVL.RB_Signal_In.HMI_STOP OR NOT GVL.RB_Signal_In.HMI_EMG OR GVL.A_RunStop 
OR POU_MONITOR_ROBOT.MC_GroupReadStatus_RBA.Error OR GVL.RB_A_.ERROR
OR SCARA_A.m_group_error > 0 THEN
	MC_Stop_A0.Execute:= TRUE;
	MC_Stop_A1.Execute:= TRUE;
	MC_Stop_A2.Execute:= TRUE;
	MC_Stop_A3.Execute:= TRUE;
	MC_GroupStop_RBA.Execute := TRUE;
ELSE
	MC_Stop_A0.Execute:= FALSE;
	MC_Stop_A1.Execute:= FALSE;
	MC_Stop_A2.Execute:= FALSE;
	MC_Stop_A3.Execute:= FALSE;
	MC_GroupStop_RBA.Execute := FALSE;
END_IF

IF Bit_Stop = TRUE OR NOT GVL.X[9] OR BitStop_Tor_B OR BitStop_Error_Axis_RB_B 
OR GVL.RB_Signal_In.HMI_STOP OR NOT GVL.RB_Signal_In.HMI_EMG 
OR POU_MONITOR_ROBOT.MC_GroupReadStatus_RBB.Error OR GVL.RB_B_.ERROR
OR SCARA_B.m_group_error > 0  THEN
	MC_Stop_B0.Execute:= TRUE;
	MC_Stop_B1.Execute:= TRUE;
	MC_Stop_B2.Execute:= TRUE;
	MC_Stop_B3.Execute:= TRUE;
	MC_GroupStop_RBB.Execute := TRUE;
ELSE
	MC_Stop_B0.Execute:= FALSE;
	MC_Stop_B1.Execute:= FALSE;
	MC_Stop_B2.Execute:= FALSE;
	MC_Stop_B3.Execute:= FALSE;
	MC_GroupStop_RBA.Execute := FALSE;
END_IF




/// Condition SoftLimit

IF GVL_1.DATA_RB_A.ENABLE_SOFT_LIMIT THEN
	DISABLE_POWER_A := 0;
	CASE ENABLE_POWER_A OF
		0:
			SMC_SetSoftwareLimits_A0.SWL_Activated := TRUE;
			SMC_SetSoftwareLimits_A1.SWL_Activated := TRUE;
			SMC_SetSoftwareLimits_A2.SWL_Activated := TRUE;
			SMC_SetSoftwareLimits_A3.SWL_Activated := TRUE;
			ENABLE_POWER_A := ENABLE_POWER_A + 5;
		5:
			SMC_SetSoftwareLimits_A0.bExecute := TRUE;
			SMC_SetSoftwareLimits_A1.bExecute := TRUE;
			SMC_SetSoftwareLimits_A2.bExecute := TRUE;
			SMC_SetSoftwareLimits_A3.bExecute := TRUE;
			ENABLE_POWER_A := ENABLE_POWER_A + 5;
		10:
			// DONE	
	END_CASE
ELSE
	ENABLE_POWER_A := 0;
	CASE DISABLE_POWER_A OF
		0:
			SMC_SetSoftwareLimits_A0.bExecute := FALSE;
			SMC_SetSoftwareLimits_A1.bExecute := FALSE;
			SMC_SetSoftwareLimits_A2.bExecute := FALSE;
			SMC_SetSoftwareLimits_A3.bExecute := FALSE;
			DISABLE_POWER_A := DISABLE_POWER_A + 5;
		5:
			SMC_SetSoftwareLimits_A0.SWL_Activated := FALSE;
			SMC_SetSoftwareLimits_A1.SWL_Activated := FALSE;
			SMC_SetSoftwareLimits_A2.SWL_Activated := FALSE;
			SMC_SetSoftwareLimits_A3.SWL_Activated := FALSE;
			DISABLE_POWER_A := DISABLE_POWER_A + 5;
		10:
			SMC_SetSoftwareLimits_A0.bExecute := TRUE;
			SMC_SetSoftwareLimits_A1.bExecute := TRUE;
			SMC_SetSoftwareLimits_A2.bExecute := TRUE;
			SMC_SetSoftwareLimits_A3.bExecute := TRUE;
			DISABLE_POWER_A := DISABLE_POWER_A + 5;			
		15:
			SMC_SetSoftwareLimits_A0.bExecute := FALSE;
			SMC_SetSoftwareLimits_A1.bExecute := FALSE;
			SMC_SetSoftwareLimits_A2.bExecute := FALSE;
			SMC_SetSoftwareLimits_A3.bExecute := FALSE;				
	END_CASE
END_IF;

/// rbB
IF GVL_1.DATA_RB_B.ENABLE_SOFT_LIMIT THEN
	DISABLE_POWER_B:= 0;
	CASE ENABLE_POWER_B OF
		0:
			SMC_SetSoftwareLimits_B0.SWL_Activated := TRUE;
			SMC_SetSoftwareLimits_B1.SWL_Activated := TRUE;
			SMC_SetSoftwareLimits_B2.SWL_Activated := TRUE;
			SMC_SetSoftwareLimits_B3.SWL_Activated := TRUE;
			ENABLE_POWER_B := ENABLE_POWER_B + 5;
		5:
			SMC_SetSoftwareLimits_B0.bExecute := TRUE;
			SMC_SetSoftwareLimits_B1.bExecute := TRUE;
			SMC_SetSoftwareLimits_B2.bExecute := TRUE;
			SMC_SetSoftwareLimits_B3.bExecute := TRUE;
			ENABLE_POWER_B := ENABLE_POWER_B + 5;
		10:
			// DONE	
	END_CASE
ELSE
	ENABLE_POWER_B := 0;
	CASE DISABLE_POWER_B OF
		0:
			SMC_SetSoftwareLimits_B0.bExecute := FALSE;
			SMC_SetSoftwareLimits_B1.bExecute := FALSE;
			SMC_SetSoftwareLimits_B2.bExecute := FALSE;
			SMC_SetSoftwareLimits_B3.bExecute := FALSE;
			DISABLE_POWER_B := DISABLE_POWER_B + 5;
		5:
			SMC_SetSoftwareLimits_B0.SWL_Activated := FALSE;
			SMC_SetSoftwareLimits_B1.SWL_Activated := FALSE;
			SMC_SetSoftwareLimits_B2.SWL_Activated := FALSE;
			SMC_SetSoftwareLimits_B3.SWL_Activated := FALSE;
			DISABLE_POWER_B := DISABLE_POWER_B + 5;
		10:
			SMC_SetSoftwareLimits_B0.bExecute := TRUE;
			SMC_SetSoftwareLimits_B1.bExecute := TRUE;
			SMC_SetSoftwareLimits_B2.bExecute := TRUE;
			SMC_SetSoftwareLimits_B3.bExecute := TRUE;
			DISABLE_POWER_B := DISABLE_POWER_B + 5;			
		15:
			SMC_SetSoftwareLimits_B0.bExecute := FALSE;
			SMC_SetSoftwareLimits_B1.bExecute := FALSE;
			SMC_SetSoftwareLimits_B2.bExecute := FALSE;
			SMC_SetSoftwareLimits_B3.bExecute := FALSE;				
	END_CASE
END_IF;
END_ACTION

END_PROGRAM

// Just_Motion_Control_x86_64_Linux_SM_WV/Application/FB_/FB_TorqueDiff
FUNCTION_BLOCK PUBLIC FB_TorqueDiff
VAR_INPUT
	Enable          : BOOL;
    TorqueNow       : INT;
	PercentVel		: INT;
    Threshold       : INT;
    CycleTime_s     : LREAL;
END_VAR
VAR_OUTPUT
	DeltaTorque     : INT;
    AbsDeltaTorque  : INT;
    TorqueSlope     : LREAL;
    Alarm           : BOOL;
END_VAR
VAR
	TorqueOld       : INT;
	VelOld			: DINT;
    FirstScan       : BOOL := TRUE;
END_VAR

// IF NOT Enable THEN
//     Alarm := FALSE;
//     DeltaTorque := 0;
//     AbsDeltaTorque := 0;
//     TorqueSlope := 0.0;
//     FirstScan := TRUE;
//     RETURN;
// END_IF;

IF FirstScan THEN
    TorqueOld := TorqueNow;
    DeltaTorque := 0;
    AbsDeltaTorque := 0;
    TorqueSlope := 0.0;
    Alarm := FALSE;
    FirstScan := FALSE;
    RETURN;
END_IF;
IF (PercentVel > 70) THEN
	DeltaTorque := TorqueNow - TorqueOld;
	AbsDeltaTorque := ABS(DeltaTorque);
END_IF;

// IF CycleTime_s > 0.0 THEN
//     TorqueSlope := DeltaTorque / CycleTime_s;
// ELSE
//     TorqueSlope := 0.0;
// END_IF;

Alarm := (AbsDeltaTorque > Threshold);

TorqueOld := TorqueNow;

END_FUNCTION_BLOCK

// Just_Motion_Control_x86_64_Linux_SM_WV/Application/PRG_ROBOT/PRG_TrackingObjectSource_A
PROGRAM PRG_TrackingObjectSource_A
VAR
    fbSensorSourceA : ARRAY[1..GVL.C_MAX_SENSOR_SOURCES] OF FB_SensorObjectSource;
    uiSensorSource : UINT;
	fbVisionSourceA : ARRAY[1..GVL.C_MAX_VISION_CHANNELS] OF FB_VisionObjectSource;
	uiVisionSource : UINT;
	fbVisionResultAdapterA : ARRAY[1..GVL.C_MAX_VISION_CHANNELS] OF FB_VisionTrackingResultAdapter;
END_VAR

VAR
    // Mỗi Vision Source có một Trigger FB độc lập để giữ TriggerID và pitch riêng.
    fbVisionTriggerA : ARRAY[1..GVL.C_MAX_VISION_CHANNELS] OF FB_VisionTrackingTrigger;

    // Camera đang xử lý trong loop.
    uiCamera : UINT;

    // Recipe TRACK_PICK hiện tại.
    uiTrackingRecipe : UINT;

    // TRUE khi Recipe/Command hiện tại cho phép Source này trigger nền.
    xTrackingVisionEnable : BOOL;

    // TRUE khi Vision Framework đã nhận đúng TriggerID đang chờ.
    xVisionCommandAccepted : BOOL;
END_VAR

//=============================================================================
// PRG_TrackingObjectSource_A
//-----------------------------------------------------------------------------
// Quản lý nhiều Sensor Source cho Tracking Queue Robot A.
// Mỗi Sensor Source có một FB riêng để giữ debounce, edge và spacing riêng.
//=============================================================================

//=============================================================================
// 1. SENSOR OBJECT SOURCES
//=============================================================================
FOR uiSensorSource := 1 TO GVL.C_MAX_SENSOR_SOURCES DO

    fbSensorSourceA[uiSensorSource](
        Enable := GVL.g_aSensorSourceConfigA[uiSensorSource].Enable,
        Reset := GVL.g_xResetTrackingObjectSourceA,
        Config := GVL.g_aSensorSourceConfigA[uiSensorSource],
        ConveyorPositionMM := REAL_TO_LREAL(GVL.g_aConveyorRuntime[1].Status.PositionMM),
        Queue := GVL.g_stTrackingQueue_A
    );

END_FOR;


//=============================================================================
// 2. VISION TRACKING BACKGROUND TRIGGER
//-----------------------------------------------------------------------------
// TRACK_PICK đang Execute sẽ mở Tracking Session.
// Chỉ Source có VisionSourceID đúng với Recipe đang chạy mới được trigger.
//=============================================================================
FOR uiVisionSource := 1 TO GVL.C_MAX_VISION_CHANNELS DO

    uiCamera := GVL.g_aVisionTrackingSourceConfigA[uiVisionSource].CameraID;
    uiTrackingRecipe := GVL.g_stMultiTrackCommandA.RecipeID;

    // Mặc định Source không được trigger.
    xTrackingVisionEnable := FALSE;

    // Chỉ bật nếu Recipe hợp lệ, command TRACK_PICK đang active và Recipe dùng Vision Source này.
    IF GVL.g_stMultiTrackCommandA.Execute
    AND uiTrackingRecipe > 0
    AND uiTrackingRecipe <= GVL.C_MAX_TRACK_RECIPES
    AND GVL.g_aMultiTrackRecipeA[uiTrackingRecipe].Enable
    AND GVL.g_aMultiTrackRecipeA[uiTrackingRecipe].ObjectSourceType = E_ObjectSourceType.VISION
    AND GVL.g_aMultiTrackRecipeA[uiTrackingRecipe].VisionSourceID = GVL.g_aVisionTrackingSourceConfigA[uiVisionSource].VisionSourceID THEN
        xTrackingVisionEnable := GVL.g_aVisionTrackingSourceConfigA[uiVisionSource].Enable;
    //END_IF;
	// Commissioning: chỉ mở Source 1 mà chưa cần TRACK_PICK.
	ELSIF GVL.g_xVisionTrackingAutoTriggerTestA AND uiVisionSource = 1 THEN
		xTrackingVisionEnable := GVL.g_aVisionTrackingSourceConfigA[uiVisionSource].Enable;
	END_IF;

    // CameraID phải hợp lệ trước khi đọc g_aVisionStatus[].
    IF xTrackingVisionEnable AND uiCamera > 0 AND uiCamera <= GVL.C_MAX_VISION_CHANNELS THEN

        // Vision xác nhận command khi CurrentTriggerID bằng TriggerID đang chờ.
        xVisionCommandAccepted := fbVisionTriggerA[uiVisionSource].WaitingAccepted
            AND GVL.g_aVisionStatus[uiCamera].CurrentTriggerID = fbVisionTriggerA[uiVisionSource].TriggerID;

        fbVisionTriggerA[uiVisionSource](
            Enable := TRUE,
            Reset := GVL.g_xResetTrackingObjectSourceA,
            Config := GVL.g_aVisionTrackingSourceConfigA[uiVisionSource],
            ConveyorPositionMM := REAL_TO_LREAL(GVL.g_aConveyorRuntime[1].Status.PositionMM),

            // TODO:
            // Thay 0.0 bằng field Velocity thực tế của ST_CONVEYOR_STATUS sau khi anh chốt tên field.
            // Trong thời gian test có thể đặt TriggerOnlyWhenMoving = FALSE.
            ConveyorVelocityMMs := GVL.g_aConveyorRuntime[1].Status.VelocityMMs,

            VisionReady := GVL.g_aVisionStatus[uiCamera].Ready,
            VisionBusy := GVL.g_aVisionStatus[uiCamera].Busy,
            CommandAccepted := xVisionCommandAccepted,
			ResultProcessedTriggerID := fbVisionSourceA[uiVisionSource].LastProcessedTriggerID
        );

        //---------------------------------------------------------------------
        // MAP TRACKING TRIGGER -> VISION COMMAND
        //---------------------------------------------------------------------
        // Execute được giữ TRUE tới khi CurrentTriggerID xác nhận đã nhận command,
        // nên Communication task 15 ms không bỏ lỡ request từ task 4 ms.
        IF fbVisionTriggerA[uiVisionSource].TriggerExecute THEN
            GVL.g_aVisionCommand[uiCamera].CameraID := uiCamera;
            GVL.g_aVisionCommand[uiCamera].JobID := GVL.g_aVisionTrackingSourceConfigA[uiVisionSource].JobID;
            GVL.g_aVisionCommand[uiCamera].Application := E_VisionApplication.VIS_APP_CONVEYOR_PICK;
            GVL.g_aVisionCommand[uiCamera].TriggerID := fbVisionTriggerA[uiVisionSource].TriggerID;
            GVL.g_aVisionCommand[uiCamera].ProductID := 0;
            GVL.g_aVisionCommand[uiCamera].CaptureConveyorPos := LREAL_TO_REAL(fbVisionTriggerA[uiVisionSource].CaptureConveyorPositionMM);
            GVL.g_aVisionCommand[uiCamera].Execute := TRUE;

        // Chỉ hạ Execute của command Tracking do chính Source này phát.
        ELSIF GVL.g_aVisionCommand[uiCamera].Application = E_VisionApplication.VIS_APP_CONVEYOR_PICK
        AND GVL.g_aVisionCommand[uiCamera].JobID = GVL.g_aVisionTrackingSourceConfigA[uiVisionSource].JobID THEN
            GVL.g_aVisionCommand[uiCamera].Execute := FALSE;
        END_IF;

    ELSE
        // Khi Source không active, reset FB để lần TRACK_PICK sau có thể trigger frame đầu ngay.
        fbVisionTriggerA[uiVisionSource](
            Enable := FALSE,
            Reset := GVL.g_xResetTrackingObjectSourceA,
            Config := GVL.g_aVisionTrackingSourceConfigA[uiVisionSource],
            ConveyorPositionMM := REAL_TO_LREAL(GVL.g_aConveyorRuntime[1].Status.PositionMM),
            ConveyorVelocityMMs := GVL.g_aConveyorRuntime[1].Status.VelocityMMs,
            VisionReady := FALSE,
            VisionBusy := FALSE,
            CommandAccepted := FALSE
        );
    END_IF;

END_FOR;


//=============================================================================
// 3. VISION RESULT ADAPTER
//-----------------------------------------------------------------------------
// Chuyển Result chung của Vision Framework thành Multi Result cho Tracking.
//=============================================================================
FOR uiVisionSource := 1 TO GVL.C_MAX_VISION_CHANNELS DO

    uiCamera := GVL.g_aVisionTrackingSourceConfigA[uiVisionSource].CameraID;

    IF uiCamera > 0 AND uiCamera <= GVL.C_MAX_VISION_CHANNELS THEN
        fbVisionResultAdapterA[uiVisionSource](
            Enable := GVL.g_aVisionTrackingSourceConfigA[uiVisionSource].Enable,
            Reset := GVL.g_xResetTrackingObjectSourceA,
            CameraID := uiCamera,
            JobID := GVL.g_aVisionTrackingSourceConfigA[uiVisionSource].JobID,
            VisionResult := GVL.g_aVisionResult[uiCamera]
        );

        // Lưu Multi Result chuẩn để Vision Object Source xử lý ở bước tiếp theo.
        GVL.g_aVisionTrackingMultiResultA[uiVisionSource] := fbVisionResultAdapterA[uiVisionSource].TrackingResult;
    END_IF;

END_FOR;


//=============================================================================
// 4. VISION OBJECT SOURCES
//-----------------------------------------------------------------------------
// Scale/Offset -> Duplicate Check -> Push Object mới vào Tracking Queue.
//=============================================================================
FOR uiVisionSource := 1 TO GVL.C_MAX_VISION_CHANNELS DO

    fbVisionSourceA[uiVisionSource](
        Enable := GVL.g_aVisionTrackingSourceConfigA[uiVisionSource].Enable,
        Reset := GVL.g_xResetTrackingObjectSourceA,
        Config := GVL.g_aVisionTrackingSourceConfigA[uiVisionSource],
        Result := GVL.g_aVisionTrackingMultiResultA[uiVisionSource],
        ConveyorPositionMM := REAL_TO_LREAL(GVL.g_aConveyorRuntime[1].Status.PositionMM),
        Queue := GVL.g_stTrackingQueue_A
    );

END_FOR;

END_PROGRAM

// Just_Motion_Control_x86_64_Linux_SM_WV/Application/FB_/ConveyorTrack/FB_SensorObjectSource
FUNCTION_BLOCK FB_SensorObjectSource
VAR_INPUT

    // Cho phép FB hoạt động.
    Enable : BOOL;

    // Reset FB.
    Reset : BOOL;

    // Cấu hình nguồn Sensor.
    Config : ST_SensorObjectSourceConfig;

    // Vị trí Conveyor hiện tại.
    ConveyorPositionMM : LREAL;

END_VAR

VAR_IN_OUT

    // Queue dùng chung.
    Queue : ST_TRACKING_QUEUE;

END_VAR

VAR_OUTPUT

    // FB đang hoạt động.
    Active : BOOL;

    // Xung một cycle khi tạo Object mới.
    NewObjectPulse : BOOL;

    // FB báo lỗi.
    Error : BOOL;

    // Mã lỗi.
    ErrorID : UDINT;

END_VAR

VAR

    // Tín hiệu Sensor chưa lọc.
    xRaw : BOOL;

    // Tín hiệu Sensor sau Debounce.
    xFiltered : BOOL;

    // Trạng thái Sensor ở cycle trước.
    xPreviousFiltered : BOOL;

    // Timer Debounce.
    tonDebounce : TON;

    // Vị trí Conveyor của lần Capture trước.
    lrLastCapturePosition : LREAL;

    // TRUE khi đã từng Capture Object.
    xHasLastCapture : BOOL;

    // Slot Queue đang kiểm tra.
    uiSlot : UINT;

END_VAR

(*
===============================================================================
FUNCTION BLOCK
    FB_SensorObjectSource

DESCRIPTION
    Tạo Object trong Queue khi Sensor phát hiện sản phẩm.

WORKFLOW
    Sensor cạnh lên
        -> Debounce
        -> Kiểm tra khoảng cách tối thiểu
        -> Tìm Slot trống
        -> Tạo Object mới
        -> Ghi vị trí Conveyor tại thời điểm Capture

NOTES
    - Sensor Source chỉ phù hợp khi vị trí ngang và góc sản phẩm đã được
      cơ khí định hướng.
    - Config.CapturePoseInConveyor là Pose mặc định tại vị trí Sensor.
===============================================================================
*)
//=============================================================================
// DEFAULT PULSE OUTPUT
//=============================================================================
NewObjectPulse := FALSE;


//=============================================================================
// RESET / DISABLE
//=============================================================================
IF Reset OR NOT Enable THEN

    Active := FALSE;

    Error := FALSE;
    ErrorID := 0;

    // Reset debounce.
    tonDebounce(IN := FALSE);

    // Reset trạng thái cạnh Sensor.
    xPreviousFiltered := FALSE;
    xFiltered := FALSE;
    xRaw := FALSE;

    // Reset lịch sử Capture.
    xHasLastCapture := FALSE;
    lrLastCapturePosition := 0.0;

    // Reset runtime tìm Slot.
    uiSlot := 0;

    // Xóa pulse.
    NewObjectPulse := FALSE;

    RETURN;

END_IF;


//=============================================================================
// ACTIVE
//=============================================================================
Active := TRUE;


//=============================================================================
// VALIDATE SENSOR CHANNEL
//=============================================================================
IF Config.DetectInputChannel = 0
OR Config.DetectInputChannel > GVL.C_MAX_DI THEN

    Error := TRUE;
    ErrorID := 9101;

    RETURN;

END_IF;


//=============================================================================
// READ AND FILTER SENSOR
//=============================================================================
xRaw :=
    GVL.X[Config.DetectInputChannel]
    = Config.DetectActiveLevel;

tonDebounce(
    IN := xRaw,
    PT := Config.DebounceTime
);

xFiltered := tonDebounce.Q;


//=============================================================================
// DETECT RISING EDGE AFTER DEBOUNCE
//=============================================================================
IF xFiltered AND NOT xPreviousFiltered THEN

    //-------------------------------------------------------------------------
    // CHECK MINIMUM OBJECT SPACING
    //-------------------------------------------------------------------------
    IF NOT xHasLastCapture
    OR ABS(ConveyorPositionMM - lrLastCapturePosition)
       >= REAL_TO_LREAL(Config.MinimumObjectSpacingMM) THEN

        //---------------------------------------------------------------------
        // FIND EMPTY QUEUE SLOT
        //---------------------------------------------------------------------
        uiSlot := 0;

        FOR uiSlot := 1 TO GVL.C_MAX_TRACK_OBJECTS DO

            IF NOT Queue.Objects[uiSlot].Valid THEN
                EXIT;
            END_IF;

        END_FOR;


        //---------------------------------------------------------------------
		// CREATE NEW OBJECT
		//---------------------------------------------------------------------
		IF uiSlot <= GVL.C_MAX_TRACK_OBJECTS THEN
		
			// Sinh ObjectID mới.
			Queue.NextObjectID := Queue.NextObjectID + 1;
		
			// Tránh ObjectID bằng 0.
			IF Queue.NextObjectID = 0 THEN
				Queue.NextObjectID := 1;
			END_IF;
		
		
			//-----------------------------------------------------------------
			// BASIC OBJECT DATA
			//-----------------------------------------------------------------
			Queue.Objects[uiSlot].Valid := TRUE;
		
			Queue.Objects[uiSlot].ObjectID :=
				Queue.NextObjectID;
		
			Queue.Objects[uiSlot].ProductClassID :=
				Config.ProductClassID;
		
		
			//-----------------------------------------------------------------
			// OBJECT SOURCE
			//-----------------------------------------------------------------
			Queue.Objects[uiSlot].SourceType :=
				E_ObjectSourceType.SENSOR;
		
			Queue.Objects[uiSlot].SourceID :=
				Config.SensorSourceID;
		
		
			//-----------------------------------------------------------------
			// CAPTURE DATA
			//-----------------------------------------------------------------
			Queue.Objects[uiSlot].PoseInConveyor :=
				Config.CapturePoseInConveyor;
		
			Queue.Objects[uiSlot].CaptureConveyorPositionMM :=
				ConveyorPositionMM;
		
			Queue.Objects[uiSlot].CurrentConveyorPositionMM :=
				ConveyorPositionMM;
		
		
			//-----------------------------------------------------------------
			// SENSOR OBJECT DEFAULT DATA
			//-----------------------------------------------------------------
			Queue.Objects[uiSlot].VisionScore := 100.0;
			Queue.Objects[uiSlot].OrientationValid := TRUE;
		
			// Sensor Source không dùng Vision metadata.
			Queue.Objects[uiSlot].TriggerID := 0;
			Queue.Objects[uiSlot].ProductID := 0;
			Queue.Objects[uiSlot].CameraID := 0;
			Queue.Objects[uiSlot].JobID := 0;
		
		
			//-----------------------------------------------------------------
			// OWNERSHIP / STATE
			//-----------------------------------------------------------------
			Queue.Objects[uiSlot].Reserved := FALSE;
			Queue.Objects[uiSlot].ReservedToolID := 0;
			Queue.Objects[uiSlot].CanPick := FALSE;
			Queue.Objects[uiSlot].AbortRequired := FALSE;
			Queue.Objects[uiSlot].MissCode := 0;
			Queue.Objects[uiSlot].ErrorID := 0;
		
			Queue.Objects[uiSlot].State :=
				E_TrackingObjectState.OBJ_DETECTED;
		
		
			//-----------------------------------------------------------------
			// QUEUE COUNT
			//-----------------------------------------------------------------
			Queue.ValidCount :=
				MIN(
					Queue.ValidCount + 1,
					GVL.C_MAX_TRACK_OBJECTS
				);
		
		
			//-----------------------------------------------------------------
			// SAVE LAST CAPTURE
			//-----------------------------------------------------------------
			lrLastCapturePosition :=
				ConveyorPositionMM;
		
			xHasLastCapture := TRUE;
			NewObjectPulse := TRUE;
		
		END_IF;

    END_IF;

END_IF;


//=============================================================================
// STORE PREVIOUS SENSOR STATE
//=============================================================================
xPreviousFiltered := xFiltered;

END_FUNCTION_BLOCK

// Just_Motion_Control_x86_64_Linux_SM_WV/Application/FB_/ConveyorTrack/FB_VisionObjectSource
FUNCTION_BLOCK FB_VisionObjectSource

VAR_INPUT
    Enable : BOOL;
    Reset : BOOL;

    Config : ST_VisionTrackingSourceConfig;

    // Kết quả đã hoàn chỉnh từ Vision Adapter.
    Result : ST_VisionTrackingMultiResult;

    // Position Conveyor hiện tại.
    ConveyorPositionMM : LREAL;
END_VAR

VAR_IN_OUT
    Queue : ST_TRACKING_QUEUE;
END_VAR

VAR_OUTPUT
    Active : BOOL;

    // Xung khi Result mới bắt đầu được xử lý.
    ResultAcceptedPulse : BOOL;

    // Xung nếu ít nhất 1 Object mới được tạo.
    NewObjectPulse : BOOL;

    AddedObjectCount : UINT;
    DuplicateCount : UINT;
    RejectedCount : UINT;

    Error : BOOL;
    ErrorID : UDINT;
	
	//=============================================================================
	// DEBUG - GIỮ TRẠNG THÁI SAU SCAN
	//=============================================================================
	LastProcessedTriggerID : UDINT;          // Trigger cuối cùng đã thực sự xử lý.
	LastProcessCode : UINT;                  // Mã bước xử lý cuối cùng.
	LastCreatedObjectID : UDINT;             // ObjectID cuối cùng đã tạo.
	LastCreatedSlot : UINT;                  // Slot Queue cuối cùng đã sử dụng.
	LastCurrentPos : ST_POS;                 // CurrentPos tại lúc tạo Object.

END_VAR

VAR
    udiLastProcessedTriggerID : UDINT;

    uiDetection : UINT;
    uiObjectCount : UINT;
    uiSlot : UINT;

    uiProductClassID : UINT;

    stPoseMM : ST_POS;
    stPoseAtCapture : ST_POS;
    stCurrentPos : ST_POS;

    lrDeltaToCurrent : LREAL;

    xDuplicate : BOOL;
END_VAR

//=============================================================================
// DEFAULT PULSE OUTPUT
//=============================================================================
ResultAcceptedPulse := FALSE;
NewObjectPulse := FALSE;
AddedObjectCount := 0;
DuplicateCount := 0;
RejectedCount := 0;


//=============================================================================
// RESET / DISABLE
//=============================================================================
IF Reset OR NOT Enable THEN
    Active := FALSE;
    Error := FALSE;
    ErrorID := 0;
    udiLastProcessedTriggerID := 0;
    uiDetection := 0;
    uiObjectCount := 0;
	
	// Xóa debug khi reset Source.
    LastProcessedTriggerID := 0;
    LastProcessCode := 0;
    LastCreatedObjectID := 0;
    LastCreatedSlot := 0;
    LastCurrentPos.X := 0.0;
    LastCurrentPos.Y := 0.0;
    LastCurrentPos.Z := 0.0;
    LastCurrentPos.A := 0.0;
	
    RETURN;
END_IF;


//=============================================================================
// ACTIVE
//=============================================================================
Active := TRUE;


//=============================================================================
// VALIDATE CONFIG
//=============================================================================
IF Config.VisionSourceID = 0 THEN
    Error := TRUE;
    ErrorID := 9201;
    RETURN;
END_IF;

IF Config.CameraID = 0
OR Config.CameraID > GVL.C_MAX_VISION_CHANNELS THEN
    Error := TRUE;
    ErrorID := 9202;
    RETURN;
END_IF;

IF Config.MaxObjectCount = 0
OR Config.MaxObjectCount > GVL.C_MAX_VISION_TRACK_OBJECTS_PER_FRAME THEN
    Error := TRUE;
    ErrorID := 9203;
    RETURN;
END_IF;


//=============================================================================
// CHỈ XỬ LÝ RESULT MỚI
//=============================================================================
IF Result.Valid
AND Result.TriggerID <> 0
AND Result.TriggerID <> udiLastProcessedTriggerID THEN

    //---------------------------------------------------------------------
    // KIỂM TRA RESULT CÓ ĐÚNG SOURCE KHÔNG
    //---------------------------------------------------------------------
//     IF Result.CameraID <> Config.CameraID
//     OR Result.JobID <> Config.JobID THEN
//         RETURN;
//     END_IF;
	
	IF Result.CameraID <> Config.CameraID THEN
		LastProcessCode := 21;    // Camera mismatch
		RETURN;
	END_IF;
	
	IF Result.JobID <> Config.JobID THEN
		LastProcessCode := 22;    // Job mismatch
		RETURN;
	END_IF;


    //---------------------------------------------------------------------
    // ĐÁNH DẤU RESULT ĐÃ NHẬN
    //---------------------------------------------------------------------
    udiLastProcessedTriggerID := Result.TriggerID;
    ResultAcceptedPulse := TRUE;
	
	// Result đã qua kiểm tra Camera/Job và được Source nhận.
	LastProcessedTriggerID := Result.TriggerID;
	LastProcessCode := 10;

    //---------------------------------------------------------------------
    // GIỚI HẠN SỐ OBJECT
    //---------------------------------------------------------------------
    uiObjectCount := Result.ObjectCount;

    IF uiObjectCount > Config.MaxObjectCount THEN
        uiObjectCount := Config.MaxObjectCount;
    END_IF;

    IF uiObjectCount > GVL.C_MAX_VISION_TRACK_OBJECTS_PER_FRAME THEN
        uiObjectCount := GVL.C_MAX_VISION_TRACK_OBJECTS_PER_FRAME;
    END_IF;


    //=========================================================================
    // DUYỆT TỪNG DETECTION
    //=========================================================================
    FOR uiDetection := 1 TO uiObjectCount DO

        //---------------------------------------------------------------------
        // DETECTION KHÔNG HỢP LỆ
        //---------------------------------------------------------------------
        IF NOT Result.Objects[uiDetection].Valid THEN
            RejectedCount := RejectedCount + 1;
			LastProcessCode := 20;

        //---------------------------------------------------------------------
        // SCORE KHÔNG ĐẠT
        //---------------------------------------------------------------------
        ELSIF Result.Objects[uiDetection].Score < Config.MinimumScore THEN
            RejectedCount := RejectedCount + 1;
			LastProcessCode := 30;

        ELSE

            //-----------------------------------------------------------------
            // PRODUCT CLASS
            //-----------------------------------------------------------------
            uiProductClassID :=
                Result.Objects[uiDetection].ProductClassID;

            IF uiProductClassID = 0 THEN
                uiProductClassID := Config.ProductClassID;
            END_IF;


            //-----------------------------------------------------------------
            // RAW -> mm
            //-----------------------------------------------------------------
            stPoseMM :=
                F_VisionTrackingRawToMM(
                    RawPos := Result.Objects[uiDetection].RawPos,
                    Config := Config
                );


            //-----------------------------------------------------------------
            // POSE TẠI THỜI ĐIỂM CAPTURE
            //
            // QUAN TRỌNG:
            // stPoseMM ở đây phải đã nằm trong CONVEYOR CS.
            //-----------------------------------------------------------------
            stPoseAtCapture := stPoseMM;

            stPoseAtCapture.X :=
                stPoseAtCapture.X + Config.VisionOffset.X;

            stPoseAtCapture.Y :=
                stPoseAtCapture.Y + Config.VisionOffset.Y;

            stPoseAtCapture.Z :=
                stPoseAtCapture.Z + Config.VisionOffset.Z;

            stPoseAtCapture.A :=
                stPoseAtCapture.A + Config.VisionOffset.A;


            //-----------------------------------------------------------------
            // ĐƯA DETECTION MỚI TỚI VỊ TRÍ CURRENT
            // Để so cùng timestamp với Queue.Objects[].CurrentPos.
            //-----------------------------------------------------------------
            lrDeltaToCurrent :=
                ConveyorPositionMM
                - Result.CaptureConveyorPositionMM;

            stCurrentPos := stPoseAtCapture;

            // Conveyor của anh đang quy ước chạy theo +X Conveyor CS.
            stCurrentPos.X :=
                stPoseAtCapture.X
                + LREAL_TO_REAL(lrDeltaToCurrent);
			
			// Lưu vị trí dùng để kiểm tra Duplicate và tạo Queue.
			LastCurrentPos := stCurrentPos;
			LastProcessCode := 35;

            //-----------------------------------------------------------------
            // DUPLICATE CHECK
            //-----------------------------------------------------------------
            xDuplicate :=
                F_IsVisionTrackingDuplicate(
                    NewCurrentPos := stCurrentPos,
                    ProductClassID := uiProductClassID,
                    Config := Config,
                    Queue := Queue
                );

            IF xDuplicate THEN
                DuplicateCount := DuplicateCount + 1;
				LastProcessCode := 40;

            ELSE

                //-------------------------------------------------------------
                // FIND EMPTY QUEUE SLOT
                //-------------------------------------------------------------
                uiSlot := 0;

                FOR uiSlot := 1 TO GVL.C_MAX_TRACK_OBJECTS DO
                    IF NOT Queue.Objects[uiSlot].Valid THEN
                        EXIT;
                    END_IF;
                END_FOR;


                //-------------------------------------------------------------
                // QUEUE FULL
                //-------------------------------------------------------------
                IF uiSlot > GVL.C_MAX_TRACK_OBJECTS THEN
                    Error := TRUE;
                    ErrorID := 9204;
					LastProcessCode := 45;
                    RETURN;
                END_IF;
				
				LastCreatedSlot := uiSlot;
				LastProcessCode := 50;

                //-------------------------------------------------------------
                // SINH OBJECT ID
                //-------------------------------------------------------------
                Queue.NextObjectID :=
                    Queue.NextObjectID + 1;

                IF Queue.NextObjectID = 0 THEN
                    Queue.NextObjectID := 1;
                END_IF;


                //-------------------------------------------------------------
                // BASIC OBJECT DATA
                //-------------------------------------------------------------
                Queue.Objects[uiSlot].Valid := TRUE;

                Queue.Objects[uiSlot].ObjectID :=
                    Queue.NextObjectID;

                Queue.Objects[uiSlot].ProductClassID :=
                    uiProductClassID;


                //-------------------------------------------------------------
                // SOURCE DATA
                //-------------------------------------------------------------
                Queue.Objects[uiSlot].SourceType :=
                    E_ObjectSourceType.VISION;

                Queue.Objects[uiSlot].SourceID :=
                    Config.VisionSourceID;


                //-------------------------------------------------------------
                // CAPTURE DATA
                //-------------------------------------------------------------
                Queue.Objects[uiSlot].PoseInConveyor :=
                    stPoseAtCapture;

                Queue.Objects[uiSlot].CaptureConveyorPositionMM :=
                    Result.CaptureConveyorPositionMM;

                Queue.Objects[uiSlot].CurrentConveyorPositionMM :=
                    ConveyorPositionMM;

                Queue.Objects[uiSlot].ConveyorOffset :=
                    LREAL_TO_REAL(lrDeltaToCurrent);

                Queue.Objects[uiSlot].CurrentPos :=
                    stCurrentPos;

                Queue.Objects[uiSlot].ConveyorCoordinate :=
                    stCurrentPos.X;


                //-------------------------------------------------------------
                // VISION DATA
                //-------------------------------------------------------------
                Queue.Objects[uiSlot].VisionPos :=
                    stPoseMM;

                Queue.Objects[uiSlot].VisionScore :=
                    Result.Objects[uiDetection].Score;

                Queue.Objects[uiSlot].OrientationValid := TRUE;

                Queue.Objects[uiSlot].TriggerID :=
                    Result.TriggerID;

                Queue.Objects[uiSlot].ProductID :=
                    Result.Objects[uiDetection].FeatureID;

                Queue.Objects[uiSlot].CameraID :=
                    Result.CameraID;

                Queue.Objects[uiSlot].JobID :=
                    Result.JobID;


                //-------------------------------------------------------------
                // OWNERSHIP / STATE
                //-------------------------------------------------------------
                Queue.Objects[uiSlot].Reserved := FALSE;
                Queue.Objects[uiSlot].ReservedToolID := 0;
                Queue.Objects[uiSlot].CanPick := FALSE;
                Queue.Objects[uiSlot].AbortRequired := FALSE;
                Queue.Objects[uiSlot].MissCode := 0;
                Queue.Objects[uiSlot].ErrorID := 0;

                Queue.Objects[uiSlot].State :=
                    E_TrackingObjectState.OBJ_DETECTED;


                //-------------------------------------------------------------
                // QUEUE COUNT
                //-------------------------------------------------------------
                Queue.ValidCount :=
                    MIN(
                        Queue.ValidCount + 1,
                        GVL.C_MAX_TRACK_OBJECTS
                    );

				// Debug latched: nếu thấy 100 nghĩa là Object chắc chắn đã được ghi vào Queue.
				LastCreatedObjectID := Queue.Objects[uiSlot].ObjectID;
				LastCreatedSlot := uiSlot;
				LastCurrentPos := Queue.Objects[uiSlot].CurrentPos;
				LastProcessCode := 100;
				
				AddedObjectCount := AddedObjectCount + 1;
				NewObjectPulse := TRUE;

            END_IF;

        END_IF;

    END_FOR;

END_IF;

END_FUNCTION_BLOCK

// Just_Motion_Control_x86_64_Linux_SM_WV/Application/FC_/Conveyor/F_VisionTrackingRawToMM
FUNCTION F_VisionTrackingRawToMM : ST_POS
VAR_INPUT
    RawPos : ST_POS;
    Config : ST_VisionTrackingSourceConfig;
END_VAR

F_VisionTrackingRawToMM := RawPos;

IF Config.ResultInPixel THEN
    F_VisionTrackingRawToMM.X := RawPos.X * Config.MMPerPixelX;
    F_VisionTrackingRawToMM.Y := RawPos.Y * Config.MMPerPixelY;
END_IF;

END_FUNCTION

// Just_Motion_Control_x86_64_Linux_SM_WV/Application/FC_/Conveyor/F_IsVisionTrackingDuplicate
FUNCTION F_IsVisionTrackingDuplicate : BOOL
VAR_INPUT
    NewCurrentPos : ST_POS;
    ProductClassID : UINT;
    Config : ST_VisionTrackingSourceConfig;
END_VAR

VAR_IN_OUT
    Queue : ST_TRACKING_QUEUE;
END_VAR

VAR
    uiObject : UINT;
    rDX : REAL;
    rDY : REAL;
    rDA : REAL;
END_VAR

F_IsVisionTrackingDuplicate := FALSE;

FOR uiObject := 1 TO GVL.C_MAX_TRACK_OBJECTS DO

    IF Queue.Objects[uiObject].Valid THEN

        //---------------------------------------------------------------------
        // Chỉ bỏ qua Object đã không còn đại diện cho vật trên Conveyor.
        //---------------------------------------------------------------------
        IF Queue.Objects[uiObject].State <> E_TrackingObjectState.OBJ_EMPTY
        AND Queue.Objects[uiObject].State <> E_TrackingObjectState.OBJ_PICKED
        AND Queue.Objects[uiObject].State <> E_TrackingObjectState.OBJ_REJECTED
        AND Queue.Objects[uiObject].State <> E_TrackingObjectState.OBJ_EXPIRED
        //AND Queue.Objects[uiObject].State <> E_TrackingObjectState.OBJ_MISSED
        AND Queue.Objects[uiObject].State <> E_TrackingObjectState.OBJ_ABORTED
        AND Queue.Objects[uiObject].State <> E_TrackingObjectState.OBJ_ERROR THEN

            //-----------------------------------------------------------------
            // ProductClass tương thích.
            //-----------------------------------------------------------------
            IF ProductClassID = 0
            OR Queue.Objects[uiObject].ProductClassID = ProductClassID THEN

                rDX := ABS(NewCurrentPos.X - Queue.Objects[uiObject].CurrentPos.X);
                rDY := ABS(NewCurrentPos.Y - Queue.Objects[uiObject].CurrentPos.Y);

                rDA := F_AngleDifferenceDeg(
                    Angle1 := NewCurrentPos.A,
                    Angle2 := Queue.Objects[uiObject].CurrentPos.A
                );

                IF rDX <= Config.DuplicateToleranceXMM
                AND rDY <= Config.DuplicateToleranceYMM
                AND rDA <= Config.DuplicateAngleDeg THEN
                    F_IsVisionTrackingDuplicate := TRUE;
                    RETURN;
                END_IF;

            END_IF;

        END_IF;

    END_IF;

END_FOR;

END_FUNCTION

// Just_Motion_Control_x86_64_Linux_SM_WV/Application/FC_/Conveyor/F_AngleDifferenceDeg
FUNCTION F_AngleDifferenceDeg : REAL
VAR_INPUT
    Angle1 : REAL;
    Angle2 : REAL;
END_VAR
VAR
    rDiff : REAL;
END_VAR

rDiff := ABS(Angle1 - Angle2);

WHILE rDiff >= 360.0 DO
    rDiff := rDiff - 360.0;
END_WHILE;

IF rDiff > 180.0 THEN
    rDiff := 360.0 - rDiff;
END_IF;

F_AngleDifferenceDeg := rDiff;

END_FUNCTION

// Just_Motion_Control_x86_64_Linux_SM_WV/Application/FB_/ConveyorTrack/FB_VisionTrackingResultAdapter
FUNCTION_BLOCK FB_VisionTrackingResultAdapter

VAR_INPUT

    // Cho phép Adapter.
    Enable : BOOL;

    // Reset Adapter.
    Reset : BOOL;

    // Camera/Source mong đợi.
    CameraID : UINT;

    // Job mong đợi.
    JobID : UINT;

    // Result chung từ Vision framework.
    VisionResult : ST_VISION_RESULT;

END_VAR


VAR_OUTPUT

    // Result chuẩn dành cho Conveyor Tracking.
    TrackingResult : ST_VisionTrackingMultiResult;

    // Xung một scan khi có Result mới hoàn chỉnh.
    NewResultPulse : BOOL;

    // Adapter đang hoạt động.
    Active : BOOL;

    // Lỗi Adapter.
    Error : BOOL;

    ErrorID : UDINT;

END_VAR


VAR

    // Trigger cuối đã xử lý.
    udiLastTriggerID : UDINT;

    // Số Object thực tế cần copy.
    uiObjectCount : UINT;

    // Index copy Object.
    uiObject : UINT;

END_VAR

//=============================================================================
// FB_VisionTrackingResultAdapter
//-----------------------------------------------------------------------------
// Chuyển ST_VISION_RESULT của Vision Framework
// thành ST_VisionTrackingMultiResult dùng cho Conveyor Tracking.
//
// Hỗ trợ:
// 1. VIS_DATA_POS          -> 1 Tracking Object.
// 2. VIS_DATA_TRACK_OBJECT -> N Tracking Objects.
//=============================================================================


//=============================================================================
// DEFAULT PULSE
//=============================================================================
NewResultPulse := FALSE;


//=============================================================================
// RESET / DISABLE
//=============================================================================
IF Reset OR NOT Enable THEN

    Active := FALSE;

    Error := FALSE;
    ErrorID := 0;

    udiLastTriggerID := 0;

    TrackingResult.Valid := FALSE;
    TrackingResult.TriggerID := 0;
    TrackingResult.CameraID := 0;
    TrackingResult.JobID := 0;
    TrackingResult.CaptureConveyorPositionMM := 0.0;
    TrackingResult.ObjectCount := 0;

    RETURN;

END_IF;


//=============================================================================
// ACTIVE
//=============================================================================
Active := TRUE;


//=============================================================================
// CHƯA CÓ RESULT HỢP LỆ
//=============================================================================
IF NOT VisionResult.Header.Valid THEN
    RETURN;
END_IF;


//=============================================================================
// KHÔNG XỬ LÝ LẠI CÙNG TRIGGER
//=============================================================================
IF VisionResult.Header.TriggerID = 0
OR VisionResult.Header.TriggerID = udiLastTriggerID THEN
    RETURN;
END_IF;


//=============================================================================
// KIỂM TRA CAMERA
//=============================================================================
IF VisionResult.Header.CameraID <> CameraID THEN

    // Không phải Result của Adapter này.
    RETURN;

END_IF;


//=============================================================================
// KIỂM TRA JOB
//=============================================================================
IF VisionResult.Header.JobID <> JobID THEN

    // Không phải Result của Job này.
    RETURN;

END_IF;


//=============================================================================
// KIỂM TRA RESULT STATUS
//=============================================================================
IF VisionResult.Header.ErrorCode <> 0 THEN

    Error := TRUE;
    ErrorID := 9211;

    // Đánh dấu Trigger đã xử lý để không báo cùng lỗi mỗi scan.
    udiLastTriggerID := VisionResult.Header.TriggerID;

    RETURN;

END_IF;


//=============================================================================
// RESET OUTPUT CHO RESULT MỚI
//=============================================================================
TrackingResult.Valid := FALSE;

TrackingResult.TriggerID :=
    VisionResult.Header.TriggerID;

TrackingResult.CameraID :=
    VisionResult.Header.CameraID;

TrackingResult.JobID :=
    VisionResult.Header.JobID;

// Quan trọng:
// Đây phải là Encoder tại lúc CAMERA CAPTURE,
// không phải Encoder tại lúc Result trả về.
TrackingResult.CaptureConveyorPositionMM :=
    REAL_TO_LREAL(VisionResult.Header.CaptureConveyorPos);

// Reset số lượng Object của frame mới.
TrackingResult.ObjectCount := 0;

// Xóa cờ Valid của dữ liệu frame trước,
// tránh monitor thấy Object cũ còn tồn tại trong Array.
FOR uiObject := 1 TO GVL.C_MAX_VISION_TRACK_OBJECTS_PER_FRAME DO
    TrackingResult.Objects[uiObject].Valid := FALSE;
END_FOR;


//=============================================================================
// XỬ LÝ THEO DATA TYPE
//=============================================================================
CASE VisionResult.Header.DataType OF


    //=========================================================================
    // MỘT POSE -> MỘT TRACKING OBJECT
    //=========================================================================
    E_VisionDataType.VIS_DATA_POS:

        IF VisionResult.PosResult.Valid THEN

            TrackingResult.ObjectCount := 1;

            TrackingResult.Objects[1].Valid := TRUE;

            TrackingResult.Objects[1].RawPos :=
                VisionResult.PosResult.Pos;

            TrackingResult.Objects[1].Score :=
                VisionResult.PosResult.Score;

            // PosResult hiện không có ProductClass.
            // VisionObjectSource sẽ lấy default từ Config.
            TrackingResult.Objects[1].ProductClassID := 0;

            TrackingResult.Objects[1].FeatureID :=
                TO_UDINT(VisionResult.PosResult.FeatureID);

            TrackingResult.Valid := TRUE;

        ELSE

            TrackingResult.ObjectCount := 0;

            // Result hợp lệ nhưng không tìm thấy Object.
            TrackingResult.Valid := TRUE;

        END_IF;


    //=========================================================================
    // N OBJECT -> N TRACKING OBJECT
    //=========================================================================
    E_VisionDataType.VIS_DATA_TRACK_OBJECT:

        //---------------------------------------------------------------------
        // Kiểm tra bộ Multi Object.
        //---------------------------------------------------------------------
        IF VisionResult.TrackObjectResult.Valid THEN

            uiObjectCount :=
                VisionResult.TrackObjectResult.ObjectCount;

            //-----------------------------------------------------------------
            // Giới hạn theo kích thước Array.
            //-----------------------------------------------------------------
            IF uiObjectCount >
                GVL.C_MAX_VISION_TRACK_OBJECTS_PER_FRAME THEN

                uiObjectCount :=
                    GVL.C_MAX_VISION_TRACK_OBJECTS_PER_FRAME;

            END_IF;


            //-----------------------------------------------------------------
            // Có thể kiểm tra thêm Header.DataCount.
            //
            // Nếu protocol quy ước:
            // Header.DataCount = số Object
            // thì lấy MIN của hai giá trị.
            //-----------------------------------------------------------------
            IF VisionResult.Header.DataCount < uiObjectCount THEN

                uiObjectCount :=
                    VisionResult.Header.DataCount;

            END_IF;


            TrackingResult.ObjectCount :=
                uiObjectCount;


            //-----------------------------------------------------------------
            // COPY TỪ VISION RESULT SANG TRACKING RESULT
            //-----------------------------------------------------------------
            FOR uiObject := 1 TO uiObjectCount DO

                TrackingResult.Objects[uiObject].Valid :=
                    VisionResult.TrackObjectResult.Objects[uiObject].Valid;

                TrackingResult.Objects[uiObject].RawPos :=
                    VisionResult.TrackObjectResult.Objects[uiObject].Pos;

                TrackingResult.Objects[uiObject].Score :=
                    VisionResult.TrackObjectResult.Objects[uiObject].Score;

                TrackingResult.Objects[uiObject].ProductClassID :=
                    VisionResult.TrackObjectResult.Objects[uiObject].ProductClassID;

                TrackingResult.Objects[uiObject].FeatureID :=
                    VisionResult.TrackObjectResult.Objects[uiObject].FeatureID;

            END_FOR;


            TrackingResult.Valid := TRUE;

        ELSE

            // Multi Object Result chưa hoàn chỉnh.
            RETURN;

        END_IF;


    //=========================================================================
    // DATA TYPE KHÁC KHÔNG PHẢI TRACKING
    //=========================================================================
    ELSE

        // Không báo Error vì Camera có thể chạy Align/Inspection/Glue.
        RETURN;

END_CASE;


//=============================================================================
// RESULT ĐÃ HOÀN THÀNH
//=============================================================================
IF TrackingResult.Valid THEN

    // Đánh dấu Trigger đã xử lý.
    udiLastTriggerID :=
        VisionResult.Header.TriggerID;

    // Xung thông báo Result mới.
    NewResultPulse := TRUE;

END_IF;

END_FUNCTION_BLOCK

// Just_Motion_Control_x86_64_Linux_SM_WV/Application/FB_/Vision/FB_VisionTrackingTrigger
FUNCTION_BLOCK FB_VisionTrackingTrigger
VAR_INPUT
    Enable : BOOL;                          // TRUE khi Tracking session cần Source này.
    Reset : BOOL;                           // Reset runtime trigger.
    Config : ST_VisionTrackingSourceConfig; // Cấu hình Source.

    ConveyorPositionMM : LREAL;             // Vị trí Conveyor hiện tại.
    ConveyorVelocityMMs : REAL;             // Tốc độ Conveyor hiện tại.

    VisionReady : BOOL;                     // Camera/Channel sẵn sàng nhận command.
    VisionBusy : BOOL;                      // Camera đang xử lý command trước.

    // TRUE khi tầng Vision framework đã nhận đúng TriggerID hiện tại.
    // Trong project hiện tại có thể nối bằng:
    // GVL.g_aVisionStatus[CameraID].CurrentTriggerID = TriggerID.
    CommandAccepted : BOOL;
	ResultProcessedTriggerID : UDINT;   // TriggerID cuối đã được VisionObjectSource xử lý.
END_VAR

VAR_OUTPUT
    TriggerExecute : BOOL;                  // Giữ TRUE tới khi CommandAccepted.
    TriggerID : UDINT;                      // ID transaction đang phát.
    CaptureConveyorPositionMM : LREAL;      // Encoder được chốt cùng TriggerID.
    Active : BOOL;                          // FB đang được Enable.
    WaitingAccepted : BOOL;                 // Đang chờ Vision nhận command.
    Error : BOOL;
    ErrorID : UDINT;
	WaitingResult : BOOL;               // Đang chờ Result của Trigger hiện tại.
END_VAR

VAR
    lrLastTriggerPositionMM : LREAL;         // Encoder của lần trigger đã được nhận gần nhất.
    xHasLastTrigger : BOOL;                  // FALSE khi chưa có trigger nào trong session.
    xRequestPending : BOOL;                  // Đã đủ điều kiện khoảng cách và đang chờ Camera Ready.
    udiNextTriggerID : UDINT;                // Bộ đếm TriggerID nội bộ Source.
END_VAR

//=============================================================================
// DEFAULT OUTPUT
//=============================================================================
TriggerExecute := WaitingAccepted;


//=============================================================================
// RESET / DISABLE
//=============================================================================
IF Reset OR NOT Enable THEN
    Active := FALSE;
    TriggerExecute := FALSE;
    WaitingAccepted := FALSE;
    Error := FALSE;
    ErrorID := 0;
    xRequestPending := FALSE;
    xHasLastTrigger := FALSE;
    lrLastTriggerPositionMM := ConveyorPositionMM;
	WaitingResult := FALSE;
    RETURN;
END_IF;

Active := TRUE;


//=============================================================================
// VALIDATE CONFIG
//=============================================================================
IF Config.TriggerPitchMM <= 0.0 THEN
    Error := TRUE;
    ErrorID := 9241;                        // TriggerPitchMM không hợp lệ.
    RETURN;
END_IF;

Error := FALSE;
ErrorID := 0;


//=============================================================================
// TẠO YÊU CẦU TRIGGER THEO QUÃNG ĐƯỜNG CONVEYOR
//-----------------------------------------------------------------------------
// Không tạo request mới khi command trước vẫn chưa được Vision nhận.
//=============================================================================
//IF Config.AutoTrigger AND NOT xRequestPending AND NOT WaitingAccepted THEN
IF Config.AutoTrigger AND NOT xRequestPending AND NOT WaitingAccepted AND NOT WaitingResult THEN
    // Nếu không bắt buộc Conveyor chạy thì bỏ qua kiểm tra Velocity.
    IF NOT Config.TriggerOnlyWhenMoving OR ABS(ConveyorVelocityMMs) >= Config.MinimumTriggerVelocityMMs THEN

        // Lần đầu khi session vừa bật: cho phép trigger ngay khi Camera Ready.
        IF NOT xHasLastTrigger THEN
            xRequestPending := TRUE;

        // Các lần tiếp theo: chỉ trigger khi Conveyor đã đi đủ TriggerPitchMM.
        ELSIF ABS(ConveyorPositionMM - lrLastTriggerPositionMM) >= REAL_TO_LREAL(Config.TriggerPitchMM) THEN
            xRequestPending := TRUE;
        END_IF;

    END_IF;

END_IF;


//=============================================================================
// PHÁT COMMAND MỚI
//-----------------------------------------------------------------------------
// TriggerID và CaptureConveyorPositionMM được chốt cùng một thời điểm.
//=============================================================================
IF xRequestPending AND VisionReady AND NOT VisionBusy AND NOT WaitingAccepted AND NOT WaitingResult THEN

    udiNextTriggerID := udiNextTriggerID + 1;
    IF udiNextTriggerID = 0 THEN udiNextTriggerID := 1; END_IF;

    TriggerID := udiNextTriggerID;
    CaptureConveyorPositionMM := ConveyorPositionMM;

    WaitingAccepted := TRUE;
    TriggerExecute := TRUE;
END_IF;


//=============================================================================
// VISION ĐÃ NHẬN COMMAND
//-----------------------------------------------------------------------------
// Chỉ khi command được nhận mới cập nhật vị trí trigger gần nhất.
// Nếu communication chậm, Execute tiếp tục được giữ TRUE qua nhiều scan.
//=============================================================================
IF WaitingAccepted AND CommandAccepted THEN
    WaitingAccepted := FALSE;
	WaitingResult := TRUE;
    TriggerExecute := FALSE;
    xRequestPending := FALSE;
    lrLastTriggerPositionMM := CaptureConveyorPositionMM;
    xHasLastTrigger := TRUE;
END_IF;

//=============================================================================
// RESULT CỦA TRIGGER HIỆN TẠI ĐÃ ĐƯỢC OBJECT SOURCE XỬ LÝ
//=============================================================================
IF WaitingResult AND TriggerID <> 0 AND ResultProcessedTriggerID = TriggerID THEN

    WaitingResult := FALSE;

END_IF;

END_FUNCTION_BLOCK

// Just_Motion_Control_x86_64_Linux_SM_WV/Application/PRG_ROBOT/PRG_TrackingQueue_A
PROGRAM PRG_TrackingQueue_A
VAR
    uiObject : UINT;
    rCurrentConveyorPos : REAL;
    rVelocityAbs : REAL;
    rDistanceToAbort : REAL;
END_VAR

//=============================================================================
// PRG_TrackingQueue_A
//-----------------------------------------------------------------------------
// Cập nhật Runtime của tất cả Object trong Tracking Queue Robot A.
//
// Nguồn vị trí Conveyor:
//     GVL.g_aConveyorRuntime[1].Status.PositionMM
//
// Chương trình này KHÔNG tạo Object.
// Sensor/Vision Source sẽ chịu trách nhiệm tạo Object ở bước sau.
//=============================================================================

rCurrentConveyorPos := GVL.g_aConveyorRuntime[1].Status.PositionMM;
rVelocityAbs := ABS(GVL.g_aConveyorRuntime[1].Status.VelocityMMs);

//=============================================================================
// CLEAR TOÀN BỘ TRACKING QUEUE
//-----------------------------------------------------------------------------
IF GVL.g_xClearTrackingQueueA THEN

    FOR uiObject := 1 TO GVL.C_MAX_TRACK_OBJECTS DO
        GVL.g_stTrackingQueue_A.Objects[uiObject].Valid := FALSE;
        GVL.g_stTrackingQueue_A.Objects[uiObject].ObjectID := 0;
        GVL.g_stTrackingQueue_A.Objects[uiObject].ProductClassID := 0;
        GVL.g_stTrackingQueue_A.Objects[uiObject].Reserved := FALSE;
        GVL.g_stTrackingQueue_A.Objects[uiObject].ReservedToolID := 0;
        GVL.g_stTrackingQueue_A.Objects[uiObject].CanPick := FALSE;
        GVL.g_stTrackingQueue_A.Objects[uiObject].AbortRequired := FALSE;
        GVL.g_stTrackingQueue_A.Objects[uiObject].State := E_TrackingObjectState.OBJ_EMPTY;
        GVL.g_stTrackingQueue_A.Objects[uiObject].MissCode := 0;
        GVL.g_stTrackingQueue_A.Objects[uiObject].ErrorID := 0;
        GVL.g_stTrackingQueue_A.Objects[uiObject].TimeRemainingSec := 0.0;
        GVL.g_stTrackingQueue_A.Objects[uiObject].ConveyorOffset := 0.0;
        GVL.g_stTrackingQueue_A.Objects[uiObject].ConveyorCoordinate := 0.0;
    END_FOR;

    GVL.g_stTrackingQueue_A.ValidCount := 0;
    GVL.g_stTrackingQueue_A.ActiveIndex := GVL.C_INVALID_INDEX;

    // Nếu muốn ObjectID quay lại từ 1 sau mỗi lần clear.
    GVL.g_stTrackingQueue_A.NextObjectID := 0;

    // Tự hạ lệnh.
    GVL.g_xClearTrackingQueueA := FALSE;

    RETURN;
END_IF;


//=============================================================================
// DUYỆT TOÀN BỘ QUEUE
//=============================================================================
FOR uiObject := 1 TO GVL.C_MAX_TRACK_OBJECTS DO

    //----------------------------------------------------------------------
    // Chỉ xử lý Slot đang có Object hợp lệ.
    //----------------------------------------------------------------------
    IF GVL.g_stTrackingQueue_A.Objects[uiObject].Valid THEN

        //------------------------------------------------------------------
        // 1. CẬP NHẬT VỊ TRÍ CONVEYOR HIỆN TẠI
        //------------------------------------------------------------------
        GVL.g_stTrackingQueue_A.Objects[uiObject].CurrentConveyorPositionMM :=
            REAL_TO_LREAL(rCurrentConveyorPos);


        //------------------------------------------------------------------
        // 2. ĐỘ DỊCH CONVEYOR TỪ THỜI ĐIỂM CAPTURE
        //------------------------------------------------------------------
        GVL.g_stTrackingQueue_A.Objects[uiObject].ConveyorOffset :=
            LREAL_TO_REAL(
                GVL.g_stTrackingQueue_A.Objects[uiObject].CurrentConveyorPositionMM
                - GVL.g_stTrackingQueue_A.Objects[uiObject].CaptureConveyorPositionMM
            );


        //------------------------------------------------------------------
        // 3. TỌA ĐỘ DỌC CONVEYOR HIỆN TẠI CỦA OBJECT
        //------------------------------------------------------------------
        // PoseInConveyor.X là tọa độ Object tại thời điểm Capture.
        GVL.g_stTrackingQueue_A.Objects[uiObject].ConveyorCoordinate :=
            GVL.g_stTrackingQueue_A.Objects[uiObject].PoseInConveyor.X
            + GVL.g_stTrackingQueue_A.Objects[uiObject].ConveyorOffset;


        //------------------------------------------------------------------
        // 4. CURRENT POS
        //------------------------------------------------------------------
        GVL.g_stTrackingQueue_A.Objects[uiObject].CurrentPos :=
            GVL.g_stTrackingQueue_A.Objects[uiObject].PoseInConveyor;

        GVL.g_stTrackingQueue_A.Objects[uiObject].CurrentPos.X :=
            GVL.g_stTrackingQueue_A.Objects[uiObject].ConveyorCoordinate;


        //------------------------------------------------------------------
        // 5. DEFAULT RUNTIME FLAGS
        //------------------------------------------------------------------
//         GVL.g_stTrackingQueue_A.Objects[uiObject].CanPick := FALSE;
//         GVL.g_stTrackingQueue_A.Objects[uiObject].AbortRequired := FALSE;
        GVL.g_stTrackingQueue_A.Objects[uiObject].TimeRemainingSec := 0.0;


//         //------------------------------------------------------------------
// 		// DEFAULT RUNTIME FLAGS
// 		//------------------------------------------------------------------
// 		GVL.g_stTrackingQueue_A.Objects[uiObject].CanPick := FALSE;
// 		GVL.g_stTrackingQueue_A.Objects[uiObject].AbortRequired := FALSE;
		
		
		//----------------------------------------------------------------------
		// OBJECT ĐÃ PICK XONG
		// Không được tính lại READY/MISSED theo vị trí Conveyor.
		//----------------------------------------------------------------------
		IF GVL.g_stTrackingQueue_A.Objects[uiObject].State
			= E_TrackingObjectState.OBJ_PICKED THEN
		
			GVL.g_stTrackingQueue_A.Objects[uiObject].CanPick := FALSE;
			GVL.g_stTrackingQueue_A.Objects[uiObject].AbortRequired := FALSE;
		
		
		//----------------------------------------------------------------------
		// OBJECT CHƯA ĐƯỢC ROBOT / TOOL SỞ HỮU
		//----------------------------------------------------------------------
		ELSIF NOT GVL.g_stTrackingQueue_A.Objects[uiObject].Reserved THEN
		
			GVL.g_stTrackingQueue_A.Objects[uiObject].CanPick := FALSE;
			GVL.g_stTrackingQueue_A.Objects[uiObject].AbortRequired := FALSE;
		
			IF GVL.g_stTrackingQueue_A.Objects[uiObject].ConveyorCoordinate
				< GVL.g_stTrackingConfig_A.Workspace.PickZoneStartMM THEN
		
				GVL.g_stTrackingQueue_A.Objects[uiObject].State :=
					E_TrackingObjectState.OBJ_WAIT_PICK_ZONE;
		
			ELSIF GVL.g_stTrackingQueue_A.Objects[uiObject].ConveyorCoordinate
				<= GVL.g_stTrackingConfig_A.Workspace.PickZoneEndMM THEN
		
				GVL.g_stTrackingQueue_A.Objects[uiObject].CanPick := TRUE;
		
				GVL.g_stTrackingQueue_A.Objects[uiObject].State :=
					E_TrackingObjectState.OBJ_READY;
		
			ELSIF GVL.g_stTrackingQueue_A.Objects[uiObject].ConveyorCoordinate
				< GVL.g_stTrackingConfig_A.Workspace.ExpirePositionMM THEN
		
				GVL.g_stTrackingQueue_A.Objects[uiObject].State :=
					E_TrackingObjectState.OBJ_MISSED;
		
			ELSE
		
				GVL.g_stTrackingQueue_A.Objects[uiObject].State :=
					E_TrackingObjectState.OBJ_EXPIRED;
		
			END_IF;
		
		
		//----------------------------------------------------------------------
		// OBJECT ĐANG ĐƯỢC TRACKING SỞ HỮU
		//----------------------------------------------------------------------
		ELSE
		
			IF GVL.g_stTrackingQueue_A.Objects[uiObject].ConveyorCoordinate
				>= GVL.g_stTrackingConfig_A.Workspace.AbortPositionMM THEN
		
				GVL.g_stTrackingQueue_A.Objects[uiObject].AbortRequired := TRUE;
		
			ELSE
		
				GVL.g_stTrackingQueue_A.Objects[uiObject].AbortRequired := FALSE;
		
			END_IF;
		
		END_IF;
		
		
		//=============================================================================
		// CLEANUP OBJECT PICKED
		//=============================================================================
		IF GVL.g_stTrackingQueue_A.Objects[uiObject].Valid
		AND NOT GVL.g_stTrackingQueue_A.Objects[uiObject].Reserved
		AND GVL.g_stTrackingQueue_A.Objects[uiObject].State
			= E_TrackingObjectState.OBJ_PICKED THEN
		
			GVL.g_stTrackingQueue_A.Objects[uiObject].Valid := FALSE;
			GVL.g_stTrackingQueue_A.Objects[uiObject].ReservedToolID := 0;
			GVL.g_stTrackingQueue_A.Objects[uiObject].CanPick := FALSE;
			GVL.g_stTrackingQueue_A.Objects[uiObject].AbortRequired := FALSE;
			GVL.g_stTrackingQueue_A.Objects[uiObject].TimeRemainingSec := 0.0;
		
			GVL.g_stTrackingQueue_A.Objects[uiObject].State :=
				E_TrackingObjectState.OBJ_EMPTY;
		
			IF GVL.g_stTrackingQueue_A.ValidCount > 0 THEN
				GVL.g_stTrackingQueue_A.ValidCount :=
					GVL.g_stTrackingQueue_A.ValidCount - 1;
			END_IF;
		
		END_IF;



// 		//------------------------------------------------------------------
// 		// OBJECT CHƯA ĐƯỢC ROBOT / TOOL SỞ HỮU
// 		//------------------------------------------------------------------
// 		IF NOT GVL.g_stTrackingQueue_A.Objects[uiObject].Reserved THEN
// 		
// 			// Queue Manager được quyền tính lại hai trạng thái này.
// 			GVL.g_stTrackingQueue_A.Objects[uiObject].CanPick := FALSE;
// 			GVL.g_stTrackingQueue_A.Objects[uiObject].AbortRequired := FALSE;
// 		
// 			// Chưa tới vùng Pick.
// 			IF GVL.g_stTrackingQueue_A.Objects[uiObject].ConveyorCoordinate
// 				< GVL.g_stTrackingConfig_A.Workspace.PickZoneStartMM THEN
// 		
// 				GVL.g_stTrackingQueue_A.Objects[uiObject].State :=
// 					E_TrackingObjectState.OBJ_WAIT_PICK_ZONE;
// 		
// 			// Đang nằm trong vùng Pick.
// 			ELSIF GVL.g_stTrackingQueue_A.Objects[uiObject].ConveyorCoordinate
// 				<= GVL.g_stTrackingConfig_A.Workspace.PickZoneEndMM THEN
// 		
// 				GVL.g_stTrackingQueue_A.Objects[uiObject].CanPick := TRUE;
// 		
// 				GVL.g_stTrackingQueue_A.Objects[uiObject].State :=
// 					E_TrackingObjectState.OBJ_READY;
// 		
// 			// Đã ra khỏi vùng Pick nhưng chưa Expire.
// 			ELSIF GVL.g_stTrackingQueue_A.Objects[uiObject].ConveyorCoordinate
// 				< GVL.g_stTrackingConfig_A.Workspace.ExpirePositionMM THEN
// 		
// 				GVL.g_stTrackingQueue_A.Objects[uiObject].State :=
// 					E_TrackingObjectState.OBJ_MISSED;
// 		
// 			// Hết hiệu lực hoàn toàn.
// 			ELSE
// 		
// 				GVL.g_stTrackingQueue_A.Objects[uiObject].State :=
// 					E_TrackingObjectState.OBJ_EXPIRED;
// 		
// 			END_IF;
// 				
// 		
// 		//------------------------------------------------------------------
// 		// OBJECT ĐÃ ĐƯỢC ROBOT / TOOL SỞ HỮU
// 		//------------------------------------------------------------------
// 		ELSE
// 		
// 			// QUAN TRỌNG:
// 			// Không thay đổi CanPick tại đây.
// 			// Object đã được chọn khi CanPick = TRUE.
// 		
// 			// Chỉ tiếp tục theo dõi điều kiện Abort.
// 			IF GVL.g_stTrackingQueue_A.Objects[uiObject].ConveyorCoordinate
// 				>= GVL.g_stTrackingConfig_A.Workspace.AbortPositionMM THEN
// 		
// 				GVL.g_stTrackingQueue_A.Objects[uiObject].AbortRequired := TRUE;
// 		
// 			ELSE
// 		
// 				GVL.g_stTrackingQueue_A.Objects[uiObject].AbortRequired := FALSE;
// 		
// 			END_IF;
// 		
// 		END_IF;


        //------------------------------------------------------------------
        // 7. TÍNH THỜI GIAN CÒN LẠI TRƯỚC ABORT
        //------------------------------------------------------------------
        IF rVelocityAbs > 0.01 THEN

            rDistanceToAbort :=
                GVL.g_stTrackingConfig_A.Workspace.AbortPositionMM
                - GVL.g_stTrackingQueue_A.Objects[uiObject].ConveyorCoordinate;

            IF rDistanceToAbort > 0.0 THEN
                GVL.g_stTrackingQueue_A.Objects[uiObject].TimeRemainingSec :=
                    rDistanceToAbort / rVelocityAbs;
            ELSE
                GVL.g_stTrackingQueue_A.Objects[uiObject].TimeRemainingSec := 0.0;
            END_IF;

        END_IF;
		
		//=============================================================================
		// CLEANUP OBJECT ĐÃ EXPIRED
		//-----------------------------------------------------------------------------
		// Object đã ra khỏi toàn bộ vùng Tracking và không còn được Tool sở hữu.
		// Giải phóng Slot để Sensor có thể sử dụng lại.
		//=============================================================================
		IF NOT GVL.g_stTrackingQueue_A.Objects[uiObject].Reserved
		AND GVL.g_stTrackingQueue_A.Objects[uiObject].State = E_TrackingObjectState.OBJ_EXPIRED THEN
		
			// Giải phóng Object.
			GVL.g_stTrackingQueue_A.Objects[uiObject].Valid := FALSE;
			GVL.g_stTrackingQueue_A.Objects[uiObject].Reserved := FALSE;
			GVL.g_stTrackingQueue_A.Objects[uiObject].ReservedToolID := 0;
		
			// Xóa trạng thái runtime.
			GVL.g_stTrackingQueue_A.Objects[uiObject].CanPick := FALSE;
			GVL.g_stTrackingQueue_A.Objects[uiObject].AbortRequired := FALSE;
			GVL.g_stTrackingQueue_A.Objects[uiObject].TimeRemainingSec := 0.0;
		
			// Đưa Slot về Empty.
			GVL.g_stTrackingQueue_A.Objects[uiObject].State :=
				E_TrackingObjectState.OBJ_EMPTY;
		
			// Giảm số Object hợp lệ trong Queue.
			IF GVL.g_stTrackingQueue_A.ValidCount > 0 THEN
				GVL.g_stTrackingQueue_A.ValidCount :=
					GVL.g_stTrackingQueue_A.ValidCount - 1;
			END_IF;
		
		END_IF;

    END_IF;

END_FOR;

END_PROGRAM

// Just_Motion_Control_x86_64_Linux_SM_WV/Application/PRG_ROBOT/PRG_MultiToolTracking_A
PROGRAM PRG_MultiToolTracking_A
VAR
    // Bộ điều phối Multi-tool.
    fbControllerA : FB_MultiToolTrackingController_A;

    // Chuẩn hóa handshake giữa Controller và Tracking Core.
    fbCoreInterfaceA : FB_TrackingCoreInterface_A;

    // Tracking Core tạo PCS, chạy Approach và thoát PCS.
    fbTrackingManagerA : FB_CONVEYOR_TRACKING_MANAGER;

    // Adapter đưg_stTrackingConfig_Aing Core vào Motion Queue Robot A.
    fbMotionAdapterA : FB_TrackingMotionQueueAdapter;

    // Chọn TCP/Tool hiện hành của AxisGroup Robot A.
    fbSelectToolA : FB_SelectRobotTool;

    // Một Tool Manager độc lập cho mỗi Tool.
    fbToolManagerA : ARRAY[0..GVL.C_MAX_TOOLS] OF FB_ToolManager;

    // Command riêng gửi tới từng Tool Manager.
    astToolCommandA : ARRAY[0..GVL.C_MAX_TOOLS] OF ST_ToolCommand;

    // Command cục bộ, tránh ghi ngược vào Command của Interpreter.
    stCommandA : ST_MultiToolTrackingCommand;

    // Gốc Conveyor dùng cho test hiện tại.
    stConveyorOriginA : MC_COORD_REF;

    // Vị trí Object cố định chỉ dùng khi test riêng Tracking Core.
    stFixedObjectPositionA : MC_COORD_REF;

    // Encoder ảo dùng khi Simulation khác SIM_OFF.
    diVirtualEncoderA : DINT;

    // Index vòng lặp Tool.
    uiTool : UINT;
	xTrackingRequestValid : BOOL;
	
	rtCreateTestObjectA : R_TRIG;
	xCoreRequestValid : BOOL;
	rtMultiTrackStartTestA : R_TRIG;
	xMultiTrackTestExecuteA : BOOL := FALSE;
	
	rtDebugCoreStartA : R_TRIG;
	rtDebugExecuteToCoreA : R_TRIG;
	rtDebugCoreRequestValidA : R_TRIG;
	
	udiDebugCoreStartCountA : UDINT;
	udiDebugExecuteToCoreCountA : UDINT;
	udiDebugCoreRequestCountA : UDINT;
	
	xDebugCoreStartLatchedA : BOOL;
	xDebugExecuteToCoreLatchedA : BOOL;
	xDebugCoreRequestLatchedA : BOOL;
	
	//=============================================================================
	// CONVEYOR RUNTIME
	//=============================================================================
	rConveyorVelocityPrevA : REAL;          // Vận tốc filtered của scan trước.
	xConveyorRuntimeFirstScanA : BOOL := TRUE; // Chống spike Acceleration khi khởi động.

	fbPower : MC_Power;
	
	// Khai bao phan tinh delta pulse moi vong quet
	count_scan, i_count, udiv, count_cal_max, count_cal : INT;
	pulse_old, pulse_track  : DINT;
	delta : REAL;
END_VAR

VAR
    rPulsePerScan : REAL;
    rFractionAcc : REAL;

    diBasePulse : DINT;
    diPulseThisScan : DINT;
    diSmoothCount : DINT;
END_VAR

IF GVL.X[8] THEN
	GVL.g_xResetTrackingObjectSourceA := TRUE;
	GVL.g_xMultiTrackResetTestA := TRUE;
	GVL.g_xClearTrackingQueueA := TRUE;
ELSE
	GVL.g_xResetTrackingObjectSourceA := FALSE;
	GVL.g_xMultiTrackResetTestA := FALSE;
	GVL.g_xClearTrackingQueueA := FALSE;
	
END_IF;

//GVL.g_axDIA[1] := GVL.X[20];


//=============================================================================
// MULTI-TOOL TRACKING TEST COMMAND
//-----------------------------------------------------------------------------
// Chỉ tạo dữ liệu Command một lần tại cạnh lên của Start Test.
// Sau này khi Interpreter hoạt động, phần này chỉ dùng cho Commissioning/Test.
//=============================================================================

rtMultiTrackStartTestA(CLK := GVL.g_xMultiTrackStartTestA);
IF rtMultiTrackStartTestA.Q THEN
    GVL.g_stMultiTrackCommandA.CommandID := GVL.g_stMultiTrackCommandA.CommandID + 1;

    IF GVL.g_stMultiTrackCommandA.CommandID = 0 THEN
        GVL.g_stMultiTrackCommandA.CommandID := 1;
    END_IF;

//     GVL.g_stMultiTrackCommandA.RecipeID := 1;
//     GVL.g_stMultiTrackCommandA.TargetPickCountOverride := 1;
//     GVL.g_stMultiTrackCommandA.ToolMaskOverride := DWORD#1;
// 
//     GVL.g_aMultiTrackRecipeA[1].Enable := TRUE;
//     GVL.g_aMultiTrackRecipeA[1].RecipeID := 1;
//     GVL.g_aMultiTrackRecipeA[1].ProductClassID := 0;
//     GVL.g_aMultiTrackRecipeA[1].TargetPickCount := 1;
//     GVL.g_aMultiTrackRecipeA[1].ToolEnableMask := DWORD#1;

	GVL.g_stMultiTrackCommandA.RecipeID := 1;
    GVL.g_stMultiTrackCommandA.TargetPickCountOverride := 1;
    GVL.g_stMultiTrackCommandA.ToolMaskOverride := DWORD#1;

    GVL.g_aMultiTrackRecipeA[1].Enable := TRUE;
    GVL.g_aMultiTrackRecipeA[1].RecipeID := 1;
    GVL.g_aMultiTrackRecipeA[1].ProductClassID := 0;
    GVL.g_aMultiTrackRecipeA[1].TargetPickCount := 1;
    GVL.g_aMultiTrackRecipeA[1].ToolEnableMask := DWORD#1;

    xMultiTrackTestExecuteA := TRUE;
END_IF;

// Khi Controller hoàn thành hoặc lỗi thì hạ Execute test.
IF GVL.g_stMultiTrackStatusA.Done OR GVL.g_stMultiTrackStatusA.Error OR GVL.g_xMultiTrackResetTestA OR GVL.g_xMultiTrackAbortTestA THEN
    xMultiTrackTestExecuteA := FALSE;
END_IF;

stCommandA := GVL.g_stMultiTrackCommandA;

stCommandA.Execute := GVL.g_stMultiTrackCommandA.Execute OR xMultiTrackTestExecuteA;

stCommandA.Reset := GVL.g_stMultiTrackCommandA.Reset OR GVL.g_xMultiTrackResetTestA;

stCommandA.Abort :=
    GVL.g_stMultiTrackCommandA.Abort
    OR GVL.g_xMultiTrackAbortTestA;


//=============================================================================
// 02. GỐC CONVEYOR VÀ OBJECT TEST
//-----------------------------------------------------------------------------
// Sau này thay stConveyorOriginA bằng cấu hình Conveyor thực tế trên HMI.
//=============================================================================
// stConveyorOriginA.X := 350.0;
// stConveyorOriginA.Y := -200.0;
// stConveyorOriginA.Z := 150.0;
// stConveyorOriginA.A := 90.0;
// stConveyorOriginA.B := 0.0;
// stConveyorOriginA.C := 0.0;

stConveyorOriginA.X := GVL.g_aConveyorRuntime[1].Config.Origin.X;
stConveyorOriginA.Y := GVL.g_aConveyorRuntime[1].Config.Origin.Y;
stConveyorOriginA.Z := GVL.g_aConveyorRuntime[1].Config.Origin.Z;
stConveyorOriginA.A := GVL.g_aConveyorRuntime[1].Config.Origin.A;
stConveyorOriginA.B := 0.0;
stConveyorOriginA.C := 0.0;

stFixedObjectPositionA := GVL.g_stTrackingSimulation.FixedObjectPosition;

// Power Axis 6
fbPower(
    Axis := AXIS_6,
    Enable := TRUE,
    bRegulatorOn := TRUE,
    bDriveStart := TRUE
);
i_count := 100;
count_cal_max := 3;
IF GVL.Y[10] <> FALSE  THEN
	IF count_scan = 0 THEN
		pulse_old := AXIS_6.diActPosition;
	END_IF
	count_scan := count_scan + 1;
	
	IF count_scan >= i_count THEN
		rPulsePerScan := TO_REAL((AXIS_6.diActPosition - pulse_old))/(i_count);
		GVL.g_HMI_PulsePerCycle_Cr := rPulsePerScan;
		count_scan := 0;
		count_cal := count_cal + 1;
	END_IF
END_IF;
udiv := udiv + 1;


IF count_cal >= count_cal_max THEN
	// Phần nguyên.
	diBasePulse := REAL_TO_DINT(TRUNC(rPulsePerScan));
	
	// Tích lũy phần lẻ.
	rFractionAcc := rFractionAcc + (rPulsePerScan - DINT_TO_REAL(diBasePulse));
	
	// Mặc định chỉ tăng phần nguyên.
	diPulseThisScan := diBasePulse;
	
	// Khi phần lẻ tích đủ 1 xung thì bù thêm 1.
	IF rFractionAcc <= -200.0 THEN
		diPulseThisScan := diPulseThisScan - 1;
		rFractionAcc := rFractionAcc + 1.0;
	END_IF;
	
	// Position đưa sang encoder trung gian.
	IF GVL.Y[10] <> FALSE THEN
		diSmoothCount := diSmoothCount + diPulseThisScan;
	END_IF
END_IF


//=============================================================================
// 03. ENCODER ẢO
//-----------------------------------------------------------------------------
// Phần này được chuyển từ PRG_ConveyorTracking cũ sang PRG mới.
//=============================================================================
IF GVL.g_stTrackingSimulation.VirtualEncoderReset THEN
    diVirtualEncoderA := 0;
ELSIF GVL.g_stTrackingSimulation.VirtualEncoderEnable THEN
    diVirtualEncoderA := diVirtualEncoderA + GVL.g_stTrackingSimulation.VirtualEncoderStepPerCycle;
END_IF;

